stStationEvents[0].aEvents[18].bFault						:= TRUE;
stStationEvents[0].aEvents[18].bEventFlag					:= NOT stMachineStatus.bSystemPowerUp AND dw_T09_EL2809.stTerminalInfo.nTerminal_State <> 8;
stStationEvents[0].aEvents[18].bEventText					:= 'T09_EL2809 card in fault' ;
stStationEvents[0].aEvents[18].sSolution					:= 'Reset System';

(*stStationEvents[0].aEvents[19].bFault						:= TRUE;
stStationEvents[0].aEvents[19].bEventFlag					:= NOT stMachineStatus.bSystemPowerUp AND dw_T10_EL2809.stTerminalInfo.nTerminal_State <> 8;
stStationEvents[0].aEvents[19].bEventText					:= 'T10_EL2809 card in fault' ;
stStationEvents[0].aEvents[19].sSolution					:= 'Reset System';*)

stStationEvents[0].aEvents[20].bFault						:= TRUE;
stStationEvents[0].aEvents[20].bEventFlag					:= NOT stMachineStatus.bSystemPowerUp AND dw_T11_EL3058.stTerminalInfo.nTerminal_State <> 8;
stStationEvents[0].aEvents[20].bEventText					:= 'T11_EL3058 card in fault' ;
stStationEvents[0].aEvents[20].sSolution					:= 'Reset System';

stStationEvents[0].aEvents[22].bFault						:= TRUE;
stStationEvents[0].aEvents[22].bEventFlag					:= NOT stMachineStatus.bSystemPowerUp AND dw_T12_EL1918.stTerminalInfo.nTerminal_State <> 8;
stStationEvents[0].aEvents[22].bEventText					:= 'T12_EL1918 card in fault' ;
stStationEvents[0].aEvents[22].sSolution					:= 'Reset System';

stStationEvents[0].aEvents[23].bFault						:= TRUE;
stStationEvents[0].aEvents[23].bEventFlag					:= NOT stMachineStatus.bSystemPowerUp AND dw_T13_EL6633.stTerminalInfo.nTerminal_State <> 8;
stStationEvents[0].aEvents[23].bEventText					:= 'T13_EL6633 card in fault' ;
stStationEvents[0].aEvents[23].sSolution					:= 'Reset System';

stStationEvents[0].aEvents[24].bFault						:= TRUE;
stStationEvents[0].aEvents[24].bEventFlag					:= bDoorClosingFlag AND (NOT dw_T05_EL1918.iLeftTouchButtonNO OR NOT dw_T05_EL1918.iRightTouchButtonNO);
stStationEvents[0].aEvents[24].bEventText					:= 'Hands out before door was closed' ;
stStationEvents[0].aEvents[24].sSolution					:= 'Reset System';

stStationEvents[0].aEvents[25].bFault						:= TRUE;
stStationEvents[0].aEvents[25].bEventFlag					:= ((stMachineStatus.eMachineState = E_MachineState.MANUAL_MODE) OR (stMachineStatus.eMachineState = E_MachineState.SYSTEM_AUTO_CYCLE ))
																AND  NOT bHMIInitialized;
stStationEvents[0].aEvents[25].bEventText					:= 'Out HMI while Machine was in Autocycle' ;
stStationEvents[0].aEvents[25].sSolution					:= 'Reset System';


stStationEvents[0].aEvents[26].bFault						:= TRUE;
stStationEvents[0].aEvents[26].bEventTimer(IN := (stMachineStatus.eMachineState = E_MachineState.SYSTEM_AUTO_CYCLE) AND NOT bAutocycleIDLE, PT := stTimers.tAutoCycleTimeOut );
stStationEvents[0].aEvents[26].bEventFlag					:= stStationEvents[0].aEvents[26].bEventTimer.Q;
stStationEvents[0].aEvents[26].bEventText					:= 'Auto Cycle Timeout' ;
stStationEvents[0].aEvents[26].sSolution					:= 'Reset System';

//STOP REQUEST

stStationEvents[0].aEvents[40].bCycleStopRequest			:= TRUE;
stStationEvents[0].aEvents[40].bEventFlag					:= NOT bHMIInitialized;
stStationEvents[0].aEvents[40].bEventText					:= 'HMI not initialized' ;
stStationEvents[0].aEvents[40].sSolution					:= '';

stStationEvents[0].aEvents[41].bCycleStopRequest			:= TRUE;
stStationEvents[0].aEvents[41].bEventTimer(IN := bAutocycleIDLE, PT := stTimers.tAutoCycleIDLETimeOut);
stStationEvents[0].aEvents[41].bEventFlag					:= stStationEvents[0].aEvents[41].bEventTimer.Q;
stStationEvents[0].aEvents[41].bEventText					:= 'Autocycle in IDLE Timeout' ;
stStationEvents[0].aEvents[41].sSolution					:= '';

stStationEvents[0].aEvents[42].bCycleStopRequest			:= TRUE;
stStationEvents[0].aEvents[42].bEventFlag					:= NOT dw_T08_EL1809.iStopButton;
stStationEvents[0].aEvents[42].bEventText					:= 'Stop Button Pressed' ;
stStationEvents[0].aEvents[42].sSolution					:= '';
END_ACTION

END_PROGRAM

// ---- POUs/MAIN.TcPOU
PROGRAM MAIN
VAR
	
 
END_VAR

A_1_PRG_Main_Master();

END_PROGRAM

// ---- POUs/C_HMI/C_1_PRG_MainHMI.TcPOU
PROGRAM C_1_PRG_MainHMI
VAR
	
	bResetTest				: BOOL;
	i						: DINT;
	n						: DINT;//TABLE INDEX

END_VAR

a_ACT_MachineStatusBaner();
b_ACT_Timers();
c_ACT_IO();

bEnableSettings				:= (stMachineStatus.eMachineState = E_MachineState.STOPPED);

stStatisticsWH[0]			:= stStatisticsHMI[0];
stStatisticsWH[1]			:= stStatisticsHMI[3];
stStatisticsWH[2]			:= stStatisticsHMI[4];

stStatisticsLT[0]			:= stStatisticsHMI[0];
stStatisticsLT[1]			:= stStatisticsHMI[1];
stStatisticsLT[2]			:= stStatisticsHMI[2];

ACTION a_ACT_MachineStatusBaner:
//Machine status banner action
//SYSTEM POWER UP
IF stMachineStatus.bSystemPowerUp THEN	
	stStatusBanner.sMachineStatusText 							:= 'SYSTEM POWER UP';	
	stStatusBanner.nMachineStatusColour 						:= nWHITE;
	stStatusBanner.nMachineStatusTxtCol 						:= nBLACK;
	stStatusBanner.sBannerBckColor 								:= sWHITE;
	stStatusBanner.sBannerTextColor 							:= sBLACK;
END_IF

(* SYSTEM INITIALISING *)
IF stMachineStatus.bInitialising THEN	
	stStatusBanner.sMachineStatusText 							:= 'SYSTEM INITIALIZING';		
	stStatusBanner.nMachineStatusColour 						:= nYELLOW;
	stStatusBanner.nMachineStatusTxtCol 						:= nBLACK;
	stStatusBanner.sBannerBckColor 								:= sYELLOW;
	stStatusBanner.sBannerTextColor 							:= sBLACK;
END_IF

(* SAFETY *)
IF stMachineStatus.bSafety THEN	
	stStatusBanner.sMachineStatusText 							:= 'SYSTEM INITIALIZING';		
	stStatusBanner.nMachineStatusColour 						:= nYELLOW;
	stStatusBanner.nMachineStatusTxtCol 						:= nBLACK;
	stStatusBanner.sBannerBckColor 								:= sYELLOW;
	stStatusBanner.sBannerTextColor 							:= sBLACK;
END_IF


(* SYSTEM READY TO START FLASH ON *)
IF stMachineStatus.bReadyToStart AND stPuls.bFlash1Hz THEN
	stStatusBanner.sMachineStatusText 							:= 'SYSTEM READY TO START';		
	stStatusBanner.nMachineStatusColour 						:= nGREEN;
	stStatusBanner.nMachineStatusTxtCol 						:= nWHITE;
	stStatusBanner.sBannerBckColor 								:= sGREEN;
	stStatusBanner.sBannerTextColor 							:= sWHITE;
ELSIF stMachineStatus.bReadyToStart AND NOT stPuls.bFlash1Hz THEN	
	stStatusBanner.sMachineStatusText 							:= 'SYSTEM READY TO START';		
	stStatusBanner.nMachineStatusColour 						:= nWHITE;
	stStatusBanner.nMachineStatusTxtCol 						:= nGREEN;
	stStatusBanner.sBannerBckColor 								:= sWHITE;
	stStatusBanner.sBannerTextColor 							:= sGREEN;
END_IF

(* SYSTEM AUTO CYCLE *)
IF stMachineStatus.bAutoCycle THEN	
	stStatusBanner.sMachineStatusText 							:= 'SYSTEM AUTO CYCLE';		
	stStatusBanner.nMachineStatusColour 						:= nGREEN;
	stStatusBanner.nMachineStatusTxtCol 						:= nWHITE;
	stStatusBanner.sBannerBckColor 								:= sGREEN;
	stStatusBanner.sBannerTextColor 							:= sWHITE;	
END_IF

(* STOPPING *)
IF stMachineStatus.bStopping AND stPuls.bFlash1Hz THEN	
	stStatusBanner.sMachineStatusText 							:= 'STOPPING';		
	stStatusBanner.nMachineStatusColour 						:= nBLACK;
	stStatusBanner.nMachineStatusTxtCol 						:= nWHITE;
	stStatusBanner.sBannerBckColor 								:= sBLACK;
	stStatusBanner.sBannerTextColor 							:= sWHITE;	
ELSIF stMachineStatus.bStopping AND NOT stPuls.bFlash1Hz THEN	
	stStatusBanner.sMachineStatusText 							:= 'STOPPING';		
	stStatusBanner.nMachineStatusColour 						:= nWHITE;
	stStatusBanner.nMachineStatusTxtCol 						:= nBLACK;
	stStatusBanner.sBannerBckColor 								:= sWHITE;
	stStatusBanner.sBannerTextColor 							:= sBLACK;	
END_IF

(*STOPPED *)
IF stMachineStatus.bStopped THEN	
	stStatusBanner.sMachineStatusText 							:= 'CYCLE STOPPED';		
	stStatusBanner.nMachineStatusColour 						:= nBLACK;
	stStatusBanner.nMachineStatusTxtCol 						:= nWHITE;
	stStatusBanner.sBannerBckColor 								:= sBLACK;
	stStatusBanner.sBannerTextColor 							:= sWHITE;	
END_IF

(* FAULT FLASH ON *)
IF stMachineStatus.bFault AND stPuls.bFlash1Hz THEN	
	stStatusBanner.sMachineStatusText 							:= 'IMMEDIATE FAULT';		
	stStatusBanner.nMachineStatusColour 						:= nRED;
	stStatusBanner.nMachineStatusTxtCol 						:= nWHITE;
	stStatusBanner.sBannerBckColor 								:= sRED;
	stStatusBanner.sBannerTextColor 							:= sWHITE;	
ELSIF stMachineStatus.bFault AND NOT stPuls.bFlash1Hz THEN	
	stStatusBanner.sMachineStatusText 							:= 'IMMEDIATE FAULT';		
	stStatusBanner.nMachineStatusColour 						:= nWHITE;
	stStatusBanner.nMachineStatusTxtCol 						:= nBLACK;
	stStatusBanner.sBannerBckColor 								:= sWHITE;
	stStatusBanner.sBannerTextColor 							:= sBLACK;	
END_IF

(* MANUAL MODE *)
IF stMachineStatus.bManualMode THEN	
	stStatusBanner.sMachineStatusText 							:= 'MANUAL MODE';		
	stStatusBanner.nMachineStatusColour 						:= nBLUE;
	stStatusBanner.nMachineStatusTxtCol 						:= nWHITE;
	stStatusBanner.sBannerBckColor 								:= sBLUE;
	stStatusBanner.sBannerTextColor 							:= sWHITE;	
END_IF
END_ACTION

ACTION b_ACT_Timers:

stTimers.tAutoCycleTimeOut		:= DINT_TO_TIME(stTimers.nAutoCycleTimeOut * 1000) ;
stTimers.tDoorOpenedSignal		:= DINT_TO_TIME(stTimers.nDoorOpenedSignal * 1000) ;
stTimers.tStation1TimeOut		:= DINT_TO_TIME(stTimers.nStation1TimeOut * 1000) ;
stTimers.tStation2TimeOut		:= DINT_TO_TIME(stTimers.nStation2TimeOut * 1000) ;
stTimers.tStation3TimeOut		:= DINT_TO_TIME(stTimers.nStation3TimeOut * 1000) ;
stTimers.tTwoHandsSignal		:= DINT_TO_TIME(stTimers.nTwoHandsSignal * 1000) ;
stTimers.tHeightTest			:= DINT_TO_TIME(stTimers.nHeightTest * 1000) ;
stTimers.tAutoCycleIDLETimeOut			:= DINT_TO_TIME(stTimers.nAutoCycleIDLETimeOut * 1000) ;
END_ACTION

ACTION c_ACT_IO:


bLeftHand							:= dw_T05_EL1918.iLeftTouchButtonNO;
bRightHand							:= dw_T05_EL1918.iRightTouchButtonNO;
END_ACTION

END_PROGRAM

// ---- POUs/B_STATIONS/B_2_HEIGHT_TEST/B_2_1_PRG_Master_Height_Test.TcPOU
PROGRAM B_2_1_PRG_Master_Height_Test

VAR

	rGoodStatistics						: ARRAY[0..1] OF  R_TRIG;
	rBadStatistics						: ARRAY[0..1] OF  R_TRIG;
	rEfficency							: STRING(510);
	
	anMinimumDistance					: ARRAY[1..3] OF REAL;
	anMaximumDistance					: ARRAY[1..3] OF REAL;

/////////////////////////////////////////////////////////////////////////////////////I O/////////////////////////////////////////////////////////////////////////////////////	
	
	abPass1								: ARRAY [1..3] OF BOOL;
	abFail1								: ARRAY [1..3] OF BOOL;
	abPass2								: ARRAY [1..3] OF BOOL;
	abFail2								: ARRAY [1..3] OF BOOL;
	tonTakeMeasure						: TON;
	abMeaurement						: ARRAY [0..1] OF BOOL;
	bMeasurementDone					: BOOL;

	abProbeError1						: ARRAY[1..4] OF BOOL;
	abProbeError2						: ARRAY[1..4] OF BOOL;
	bGeneralProbeError					: BOOL;
	bGeneralError						: BOOL;
	anRawMesurement1					: ARRAY[1..4] OF REAL;
	anRawMesurement2					: ARRAY[1..4] OF REAL;
	anRealDistance1						: ARRAY[1..3] OF REAL;
	anRealDistance2						: ARRAY[1..3] OF REAL;
	

	
	i									: DINT;
	j									: DINT; //Index for settings
	
	
	

	
END_VAR

d_ACT_Set_Events_Station_2();
a_ACT_Ctrl_Station_2();
b_ACT_IO();
c_ACT_Statistics_Station_2();
e_ACT_Measurement();
f_ACT_ManualMode();
g_ACT_Settings();

ACTION a_ACT_Ctrl_Station_2:
/////////////////////////////////////////////////////////////////////////////////////UTILITIES/////////////////////////////////////////////////////////////////////////////////////
IF bGeneralProbeError OR bGeneralError OR stHeightTests.CMD.bAbort THEN
	
	stHeightTests.State			:= E_HeightTest_State.RESET;

ELSIF stHeightTests.CMD.bManualMode THEN
	
	stHeightTests.State			:= E_HeightTest_State.MANUAL_MODE;
	
END_IF



/////////////////////////////////////////////////////////////////////////////////////CONDITIONS/////////////////////////////////////////////////////////////////////////////////////

CASE stHeightTests.State OF
	
	E_HeightTest_State.ABORTED:

								IF 	stHeightTests.CMD.bEnable THEN
									
									stHeightTests.State			:= E_HeightTest_State.READY;
								
								END_IF
								
								

	E_HeightTest_State.READY:
	
								IF stHeightTests.CMD.bExecute THEN
									
									stHeightTests.State			:= E_HeightTest_State.MEASURE;
								
								END_IF
		
	E_HeightTest_State.MEASURE:				
									
								IF stHeightTests.CMD.HeightTest_CMD.Measurement1 AND stHeightTests.CMD.HeightTest_CMD.Measurement2 THEN
										
									abMeaurement[0]			:= TRUE;
									abMeaurement[1]			:= TRUE;
									
								ELSIF stHeightTests.CMD.HeightTest_CMD.Measurement1 AND NOT stHeightTests.CMD.HeightTest_CMD.Measurement2 THEN
									
									abMeaurement[0]			:= TRUE;
									
								ELSIF NOT stHeightTests.CMD.HeightTest_CMD.Measurement1 AND stHeightTests.CMD.HeightTest_CMD.Measurement2 THEN
									
									abMeaurement[1]			:= TRUE;
									
								END_IF
									
								stHeightTests.State			:= E_HeightTest_State.WAIT_MEASUREMENT;
								
	E_HeightTest_State.WAIT_MEASUREMENT:						
								
								e_ACT_Measurement();
								
								IF stHeightTests.CMD.HeightTest_CMD.Measurement1 THEN
									
									stCycleDataNest1.HeightTest_anRawMeasurement				:= anRawMesurement1;
									stCycleDataNest1.HeightTest_anDistancesResult 				:= anRealDistance1;
									stCycleDataNest1.HeightTest_bDistancesResult				:= abPass1;
									
								END_IF
								IF stHeightTests.CMD.HeightTest_CMD.Measurement2 THEN
									
									stCycleDataNest2.HeightTest_anRawMeasurement				:= anRawMesurement2;																
									stCycleDataNest2.HeightTest_anDistancesResult 				:= anRealDistance2;																
									stCycleDataNest2.HeightTest_bDistancesResult				:= abPass2;
									
								END_IF
								
								
								IF bMeasurementDone THEN
			
									stHeightTests.State		:= E_HeightTest_State.DONE;
								
								END_IF
										
	E_HeightTest_State.DONE:
								IF  stHeightTests.CMD.bAcknowledge THEN
									
									stHeightTests.State									:= E_HeightTest_State.RESULTS;
									stHeightTests.CMD.bAcknowledge 						:= FALSE;
									
								END_IF	
								
	E_HeightTest_State.RESULTS:
							
								IF abMeaurement[0] THEN
									IF abPass1[1] AND abPass1[2] AND abPass1[3] THEN
									
										stCycleDataNest1.HeightTest_Pass				:= TRUE;
									
									ELSE stCycleDataNest1.HeightTest_Fail 				:= TRUE;
								
									END_IF
								END_IF
								
								IF abMeaurement[1] THEN
									IF abPass2[1] AND abPass2[2] AND abPass2[3] THEN
									
										stCycleDataNest2.HeightTest_Pass				:= TRUE;
									
									ELSE stCycleDataNest2.HeightTest_Fail  			:= TRUE;
								
									END_IF
								END_IF	
								
								stHeightTests.State										:= E_HeightTest_State.RESET;
								
	E_HeightTest_State.RESET:
	
								abMeaurement[0]											:= FALSE;
								abMeaurement[1]											:= FALSE;
								bMeasurementDone										:= FALSE;

								FOR i := 1 TO 3 DO
									
									abPass1[i]											:= FALSE;
									abFail1[i]											:= FALSE;
									abPass2[i]											:= FALSE;
									abFail2[i]											:= FALSE;
								
								END_FOR
								
								IF bGeneralProbeError OR bGeneralError THEN
									
									stHeightTests.State									:= E_HeightTest_State.ERROR;
								
								ELSIF stHeightTests.CMD.bAbort THEN
									
									stHeightTests.State									:= E_HeightTest_State.ABORTED;
								
								ELSE stHeightTests.State								:= E_HeightTest_State.READY;
									
								END_IF
								
								
	
	E_HeightTest_State.ERROR:
	
								IF NOT bGeneralProbeError OR bGeneralError THEN
									
									stHeightTests.State									:= E_HeightTest_State.RESET;
									
								END_IF
							
	E_HeightTest_State.MANUAL_MODE:
	
								f_ACT_ManualMode();
								
								IF NOT stHeightTests.CMD.bManualMode THEN
									
									stHeightTests.State									:= E_HeightTest_State.ABORTED;
									
								END_IF
								
	
								

ELSE stHeightTests.State := E_HeightTest_State.READY;
	
END_CASE
/////////////////////////////////////////////////////////////////////////////////////STATUS/////////////////////////////////////////////////////////////////////////////////////

stHeightTests.Status.bBusy	:= 	stHeightTests.State	= E_HeightTest_State.WAIT_MEASUREMENT;	

stHeightTests.Status.bDone	:= 	stHeightTests.State	= E_HeightTest_State.DONE;

stHeightTests.Status.bError	:= 	stHeightTests.State	= E_HeightTest_State.ERROR;	

stHeightTests.Status.bReady	:=	stHeightTests.State	= E_HeightTest_State.READY;

stHeightTests.Status.bStopped := NOT stHeightTests.Status.bBusy;
END_ACTION

ACTION b_ACT_IO:

	abProbeError1					:= Probes.stProbesSet[1].abProbeError;
	abProbeError2					:= Probes.stProbesSet[2].abProbeError;
	bGeneralError					:= Probes.bGeneralError;
	anRawMesurement1				:= Probes.stProbesSet[1].anScaledRawMeasurement;
	anRawMesurement2				:= Probes.stProbesSet[2].anScaledRawMeasurement;
	


	bGeneralProbeError				:= 	abProbeError1[1] OR abProbeError1[2] OR abProbeError1[3] OR abProbeError1[4] OR
										abProbeError2[1] OR abProbeError2[2] OR abProbeError2[3] OR abProbeError2[4];
										
	stCycleDataNest1.HeightTest_anSetPoint := stProbesSettings.anExpectedDistances;
	stCycleDataNest2.HeightTest_anSetPoint := stProbesSettings.anExpectedDistances;
END_ACTION

ACTION c_ACT_Statistics_Station_2:
stStatisticsHMI[3].sName			:= 'Height Test 1';
stStatisticsHMI[4].sName			:= 'Height Test 2';


rGoodStatistics[0]( CLK := stCycleDataNest1.HeightTest_Pass);
rGoodStatistics[1]( CLK := stCycleDataNest2.HeightTest_Pass);
rBadStatistics[0]	( CLK := stCycleDataNest1.HeightTest_Fail);
rBadStatistics[1]	( CLK := stCycleDataNest2.HeightTest_Fail);

//statistics 1
IF 	rGoodStatistics[0].Q THEN
	
	stStatisticsHMI[3].nGood		:= stStatisticsHMI[3].nGood + 1;
	stStatisticsHMI[3].nTotalGood	:= stStatisticsHMI[3].nTotalGood + 1;
	
END_IF
								
IF 	rBadStatistics[0].Q THEN
	
	stStatisticsHMI[3].nBad			:= stStatisticsHMI[3].nBad + 1;
	stStatisticsHMI[3].nTotalBad	:= stStatisticsHMI[3].nTotalBad + 1;
	
END_IF

IF stStatisticsHMI[3].bResetGood THEN
	stStatisticsHMI[3].nGood		:= 0;
END_IF

IF stStatisticsHMI[3].bResetBad THEN
	stStatisticsHMI[3].nBad			:= 0;
END_IF

IF (( stStatisticsHMI[3].nGood + stStatisticsHMI[3].nBad) <> 0) THEN
	
	rEfficency							:= LREAL_TO_FMTSTR(in := (DINT_TO_REAL(stStatisticsHMI[3].nGood) /( DINT_TO_REAL(stStatisticsHMI[3].nGood) + DINT_TO_REAL(stStatisticsHMI[3].nBad))) * 100.0,iPrecision := 2, bRound := TRUE);
	stStatisticsHMI[3].nEfficency		:= CONCAT(STR1 := '%', STR2 := (rEfficency));

ELSE stStatisticsHMI[3].nEfficency		:= CONCAT(STR1 := '%', STR2 := (DINT_TO_STRING(0)));
	
END_IF
//statistics 2
IF 	rGoodStatistics[1].Q THEN
	
	stStatisticsHMI[4].nGood		:= stStatisticsHMI[4].nGood + 1;
	stStatisticsHMI[4].nTotalGood	:= stStatisticsHMI[4].nTotalGood + 1;
	
END_IF
								
IF 	rBadStatistics[1].Q THEN
	
	stStatisticsHMI[4].nBad			:= stStatisticsHMI[4].nBad + 1;
	stStatisticsHMI[4].nTotalBad	:= stStatisticsHMI[4].nTotalBad + 1;
	
END_IF

IF stStatisticsHMI[4].bResetGood THEN
	stStatisticsHMI[4].nGood		:= 0;
END_IF

IF stStatisticsHMI[4].bResetBad THEN
	stStatisticsHMI[4].nBad			:= 0;
END_IF

IF (( stStatisticsHMI[4].nGood + stStatisticsHMI[4].nBad) <> 0) THEN
	
	rEfficency							:= LREAL_TO_FMTSTR(in := (DINT_TO_REAL(stStatisticsHMI[4].nGood) /( DINT_TO_REAL(stStatisticsHMI[4].nGood) + DINT_TO_REAL(stStatisticsHMI[4].nBad))) * 100.0,iPrecision := 2, bRound := TRUE);
	stStatisticsHMI[4].nEfficency		:= CONCAT(STR1 := '%', STR2 := (rEfficency));

ELSE stStatisticsHMI[4].nEfficency		:= CONCAT(STR1 := '%', STR2 := (DINT_TO_STRING(0)));
	
END_IF
END_ACTION

ACTION d_ACT_Set_Events_Station_2:
//FAULTS

stStationEvents[2].aEvents[0].bFault						:= TRUE;
stStationEvents[2].aEvents[0].bEventFlag					:= bGeneralError;
stStationEvents[2].aEvents[0].bEventText					:= 'Probes general error';
stStationEvents[2].aEvents[0].sSolution						:= 'Check probes amplifier and ethercat unit';

stStationEvents[2].aEvents[1].bFault						:= TRUE;
stStationEvents[2].aEvents[1].bEventFlag					:= abProbeError1[1];
stStationEvents[2].aEvents[1].bEventText					:= 'Probes 1 error';
stStationEvents[2].aEvents[1].sSolution						:= 'Check probe 1';

stStationEvents[2].aEvents[2].bFault						:= TRUE;
stStationEvents[2].aEvents[2].bEventFlag					:= abProbeError1[2];
stStationEvents[2].aEvents[2].bEventText					:= 'Probes 2 error';
stStationEvents[2].aEvents[2].sSolution						:= 'Check probe 2';

stStationEvents[2].aEvents[3].bFault						:= TRUE;
stStationEvents[2].aEvents[3].bEventFlag					:= abProbeError1[3];
stStationEvents[2].aEvents[3].bEventText					:= 'Probes 3 error';
stStationEvents[2].aEvents[3].sSolution						:= 'Check probe 3';

stStationEvents[2].aEvents[4].bFault						:= TRUE;
stStationEvents[2].aEvents[4].bEventFlag					:= abProbeError1[4];
stStationEvents[2].aEvents[4].bEventText					:= 'Probes 4 error';
stStationEvents[2].aEvents[4].sSolution						:= 'Check probe 4';

stStationEvents[2].aEvents[5].bFault						:= TRUE;
stStationEvents[2].aEvents[5].bEventFlag					:= abProbeError2[1];
stStationEvents[2].aEvents[5].bEventText					:= 'Probes 5 error';
stStationEvents[2].aEvents[5].sSolution						:= 'Check probe 5';

stStationEvents[2].aEvents[6].bFault						:= TRUE;
stStationEvents[2].aEvents[6].bEventFlag					:= abProbeError2[2];
stStationEvents[2].aEvents[6].bEventText					:= 'Probes 6 error';
stStationEvents[2].aEvents[6].sSolution						:= 'Check probe 6';

stStationEvents[2].aEvents[7].bFault						:= TRUE;
stStationEvents[2].aEvents[7].bEventFlag					:= abProbeError2[3];
stStationEvents[2].aEvents[7].bEventText					:= 'Probes 7 error';
stStationEvents[2].aEvents[7].sSolution						:= 'Check probe 7';

stStationEvents[2].aEvents[8].bFault						:= TRUE;
stStationEvents[2].aEvents[8].bEventFlag					:= abProbeError2[4];
stStationEvents[2].aEvents[8].bEventText					:= 'Probes 8 error';
stStationEvents[2].aEvents[8].sSolution						:= 'Check probe 8';

stStationEvents[2].aEvents[9].bFault						:= TRUE;
stStationEvents[2].aEvents[9].bEventTimer(IN := stHeightTests.Status.bBusy, PT := stTimers.tStation2TimeOut);
stStationEvents[2].aEvents[9].bEventFlag					:= stStationEvents[2].aEvents[9].bEventTimer.Q;
stStationEvents[2].aEvents[9].bEventText					:= 'Height test cycle Timeout';
stStationEvents[2].aEvents[9].sSolution						:= 'Reset System';

(*//CYCLE STOP FAULT

stStationEvents[2].aEvents[1].bFault						:= TRUE;
stStationEvents[2].aEvents[1].bEventFlag					:= bEventsFlag[1];
stStationEvents[2].aEvents[1].bEventText					:= 'ST1 EVENT 1';
stStationEvents[2].aEvents[1].sSolution						:= 'Solution 4';


//CYCLE STOP REQUEST

stStationEvents[2].aEvents[2].bCycleStopRequest				:= TRUE;
stStationEvents[2].aEvents[2].bEventFlag					:= bEventsFlag[2];
stStationEvents[2].aEvents[2].bEventText					:= 'ST1 EVENT 2';*)
END_ACTION

ACTION e_ACT_Measurement:

tonTakeMeasure(IN:= stHeightTests.State = E_HeightTest_State.WAIT_MEASUREMENT, PT := stTimers.tHeightTest);

IF tonTakeMeasure.Q THEN
	
	IF abMeaurement[0] THEN
	
		FOR i := 1 TO 3 DO
		
			IF (anRealDistance1[i] > anMinimumDistance[i]) AND (anRealDistance1[i] < anMaximumDistance[i]) THEN
		
				abPass1[i]						:= TRUE;
			
			ELSE abFail1[i]						:= TRUE;	
				
			END_IF
		
		END_FOR

	END_IF
	
	IF abMeaurement[1] THEN
	
		FOR i := 1 TO 3 DO
		
			IF (anRealDistance2[i] > anMinimumDistance[i]) AND (anRealDistance2[i] < anMaximumDistance[i]) THEN
		
				abPass2[i]						:= TRUE;
			
			ELSE abFail2[i]						:= TRUE;	
				
			END_IF
		
		END_FOR

	END_IF

	bMeasurementDone							:= TRUE;
	i											:= 0;
END_IF
END_ACTION

ACTION f_ACT_ManualMode:
IF stPuls.bFlash100Hz THEN
	
	FOR i := 1 TO 3 DO
		
		IF (anRealDistance1[i] > anMinimumDistance[i]) AND (anRealDistance1[i] < anMaximumDistance[i]) THEN
		
			stAnimations.abDistanceBoxesGreen[i]	:= TRUE;
			
		ELSE stAnimations.abDistanceBoxesGreen[i]	:= FALSE;	
				
		END_IF
		
	END_FOR
	i												:= 0;
	FOR i := 1 TO 3 DO
		
		IF (anRealDistance2[i] > anMinimumDistance[i]) AND (anRealDistance2[i] < anMaximumDistance[i]) THEN
		
			stAnimations.abDistanceBoxesGreen[3+i]	:= TRUE;
			
		ELSE stAnimations.abDistanceBoxesGreen[3+i]	:= FALSE;	
				
		END_IF
		
	END_FOR
	
	i												:= 0;
END_IF
END_ACTION

ACTION g_ACT_Settings:
//settings tolerances

anMinimumDistance[1]					:= stProbesSettings.anExpectedDistances[1] - stProbesSettings.anTolerances[1];//settings from HMI
anMaximumDistance[1]					:= stProbesSettings.anExpectedDistances[1] + stProbesSettings.anTolerances[1];//settings from HMI
anMinimumDistance[2]					:= stProbesSettings.anExpectedDistances[2] - stProbesSettings.anTolerances[2];//settings from HMI
anMaximumDistance[2]					:= stProbesSettings.anExpectedDistances[2] + stProbesSettings.anTolerances[2];//settings from HMI
anMinimumDistance[3]					:= stProbesSettings.anExpectedDistances[3] - stProbesSettings.anTolerances[3];//settings from HMI
anMaximumDistance[3]					:= stProbesSettings.anExpectedDistances[3] + stProbesSettings.anTolerances[3];//settings from HMI





//setting the bit according to the probe from bit 1 to bit 8
IF abPresetProbe[1] THEN
	
	Probes.abPresetProbe						:= 2;

ELSIF abPresetProbe[2] THEN
	
	Probes.abPresetProbe						:= 4;
	
ELSIF abPresetProbe[3] THEN
	
	Probes.abPresetProbe						:= 8;
	
ELSIF abPresetProbe[4] THEN
	
	Probes.abPresetProbe						:= 16;
	
ELSIF abPresetProbe[5] THEN
	
	Probes.abPresetProbe						:= 32;
	
ELSIF abPresetProbe[6] THEN
	
	Probes.abPresetProbe						:= 64;
	
ELSIF abPresetProbe[7] THEN
	
	Probes.abPresetProbe						:= 128;
	
ELSIF abPresetProbe[8] THEN
	
	Probes.abPresetProbe						:= 256;

END_IF

Probes.stProbesSet[1].anScaledRawMeasurement[1]					:= DINT_TO_REAL(Probes.stProbesSet[1].anRawMeasurement[1])/10000;
Probes.stProbesSet[1].anScaledRawMeasurement[2]					:= DINT_TO_REAL(Probes.stProbesSet[1].anRawMeasurement[2])/10000;
Probes.stProbesSet[1].anScaledRawMeasurement[3]					:= DINT_TO_REAL(Probes.stProbesSet[1].anRawMeasurement[3])/10000;
Probes.stProbesSet[1].anScaledRawMeasurement[4]					:= DINT_TO_REAL(Probes.stProbesSet[1].anRawMeasurement[4])/10000;

Probes.stProbesSet[2].anScaledRawMeasurement[1]					:= DINT_TO_REAL(Probes.stProbesSet[2].anRawMeasurement[1])/10000;
Probes.stProbesSet[2].anScaledRawMeasurement[2]					:= DINT_TO_REAL(Probes.stProbesSet[2].anRawMeasurement[2])/10000;
Probes.stProbesSet[2].anScaledRawMeasurement[3]					:= DINT_TO_REAL(Probes.stProbesSet[2].anRawMeasurement[3])/10000;
Probes.stProbesSet[2].anScaledRawMeasurement[4]					:= DINT_TO_REAL(Probes.stProbesSet[2].anRawMeasurement[4])/10000;

IF Probes.stProbesSet[1].anScaledRawMeasurement[1] > 4 AND Probes.stProbesSet[1].anScaledRawMeasurement[1] < 8 AND 
	Probes.stProbesSet[1].anScaledRawMeasurement[2] > 4 AND Probes.stProbesSet[1].anScaledRawMeasurement[2] < 8 AND 
	Probes.stProbesSet[1].anScaledRawMeasurement[3] > 4 AND Probes.stProbesSet[1].anScaledRawMeasurement[3] < 8 AND 
	Probes.stProbesSet[1].anScaledRawMeasurement[4] > 4 AND Probes.stProbesSet[1].anScaledRawMeasurement[4] < 8 THEN 
	
	bEnableSetCablibrationBlock1								:= TRUE;
	
ELSE bEnableSetCablibrationBlock1								:= FALSE;
	
END_IF

IF Probes.stProbesSet[2].anScaledRawMeasurement[1] > 4 AND Probes.stProbesSet[2].anScaledRawMeasurement[1] < 8 AND 
	Probes.stProbesSet[2].anScaledRawMeasurement[2] > 4 AND Probes.stProbesSet[2].anScaledRawMeasurement[2] < 8 AND 
	Probes.stProbesSet[2].anScaledRawMeasurement[3] > 4 AND Probes.stProbesSet[2].anScaledRawMeasurement[3] < 8 AND 
	Probes.stProbesSet[2].anScaledRawMeasurement[4] > 4 AND Probes.stProbesSet[2].anScaledRawMeasurement[4] < 8 THEN 
	
	bEnableSetCablibrationBlock2								:= TRUE;
	
ELSE bEnableSetCablibrationBlock2								:= FALSE;
	
END_IF

//calibration block
IF bSetCalibrationBlock1 THEN
	
	stProbesSettings.anHeightSetByCalibration1[1]				:= Probes.stProbesSet[1].anScaledRawMeasurement[1];
	stProbesSettings.anHeightSetByCalibration1[2]				:= Probes.stProbesSet[1].anScaledRawMeasurement[2];
	stProbesSettings.anHeightSetByCalibration1[3]				:= Probes.stProbesSet[1].anScaledRawMeasurement[3];
	stProbesSettings.anHeightSetByCalibration1[4]				:= Probes.stProbesSet[1].anScaledRawMeasurement[4];
	
	stProbesSettings.nDistanceOffset1[1]						:= stProbesSettings.anDistanceCalibrationBlock[1] - (Probes.stProbesSet[1].anScaledRawMeasurement[2] - Probes.stProbesSet[1].anScaledRawMeasurement[1]);
	stProbesSettings.nDistanceOffset1[2]						:= stProbesSettings.anDistanceCalibrationBlock[2] - (Probes.stProbesSet[1].anScaledRawMeasurement[3] - Probes.stProbesSet[1].anScaledRawMeasurement[1]);
	stProbesSettings.nDistanceOffset1[3]						:= stProbesSettings.anDistanceCalibrationBlock[3] - (Probes.stProbesSet[1].anScaledRawMeasurement[4] - Probes.stProbesSet[1].anScaledRawMeasurement[1]);
	
END_IF

IF bSetCalibrationBlock2 THEN
	
	stProbesSettings.anHeightSetByCalibration2[1]				:= Probes.stProbesSet[2].anScaledRawMeasurement[1];
	stProbesSettings.anHeightSetByCalibration2[2]				:= Probes.stProbesSet[2].anScaledRawMeasurement[2];
	stProbesSettings.anHeightSetByCalibration2[3]				:= Probes.stProbesSet[2].anScaledRawMeasurement[3];
	stProbesSettings.anHeightSetByCalibration2[4]				:= Probes.stProbesSet[2].anScaledRawMeasurement[4];
	
	stProbesSettings.nDistanceOffset2[1]						:= stProbesSettings.anDistanceCalibrationBlock[1] - (Probes.stProbesSet[2].anScaledRawMeasurement[2] - Probes.stProbesSet[2].anScaledRawMeasurement[1]);
	stProbesSettings.nDistanceOffset2[2]						:= stProbesSettings.anDistanceCalibrationBlock[2] - (Probes.stProbesSet[2].anScaledRawMeasurement[3] - Probes.stProbesSet[2].anScaledRawMeasurement[1]);
	stProbesSettings.nDistanceOffset2[3]						:= stProbesSettings.anDistanceCalibrationBlock[3] - (Probes.stProbesSet[2].anScaledRawMeasurement[4] - Probes.stProbesSet[2].anScaledRawMeasurement[1]);

END_IF

anRealDistance1[1] 								:= (Probes.stProbesSet[1].anScaledRawMeasurement[2] - Probes.stProbesSet[1].anScaledRawMeasurement[1]) + stProbesSettings.nDistanceOffset1[1];
anRealDistance1[2] 								:= (Probes.stProbesSet[1].anScaledRawMeasurement[3] - Probes.stProbesSet[1].anScaledRawMeasurement[1]) + stProbesSettings.nDistanceOffset1[2];
anRealDistance1[3] 								:= (Probes.stProbesSet[1].anScaledRawMeasurement[4] - Probes.stProbesSet[1].anScaledRawMeasurement[1]) + stProbesSettings.nDistanceOffset1[3];

anRealDistance2[1] 								:= (Probes.stProbesSet[2].anScaledRawMeasurement[2] - Probes.stProbesSet[2].anScaledRawMeasurement[1]) + stProbesSettings.nDistanceOffset2[1];
anRealDistance2[2] 								:= (Probes.stProbesSet[2].anScaledRawMeasurement[3] - Probes.stProbesSet[2].anScaledRawMeasurement[1]) + stProbesSettings.nDistanceOffset2[2];
anRealDistance2[3] 								:= (Probes.stProbesSet[2].anScaledRawMeasurement[4] - Probes.stProbesSet[2].anScaledRawMeasurement[1]) + stProbesSettings.nDistanceOffset2[3];
END_ACTION

END_PROGRAM

// ---- POUs/B_STATIONS/B_1_LEAK_TEST/B_1_1_PRG_Master_Leak_Test.TcPOU
PROGRAM B_1_1_PRG_Master_Leak_Test

VAR

	tonStationStopped					: TON;
	tonExecute							: TON;
	rGoodStatistics						: ARRAY [0..1] OF R_TRIG;
	rBadStatistics						: ARRAY [0..1] OF R_TRIG;
	rEfficency							: ARRAY [0..1] OF STRING(510);
	
	tonWaitResults						: TON;
/////////////////////////////////////////////////////////////////////////////////////I O/////////////////////////////////////////////////////////////////////////////////////	

	bStopped							: ARRAY [0..1] OF BOOL;
	bError								: ARRAY [0..1] OF BOOL;
	bReady								: ARRAY [0..1] OF BOOL;
	bDone								: ARRAY [0..1] OF BOOL;
	bReset								: ARRAY [0..1] OF BOOL;
	bStart								: ARRAY [0..1] OF BOOL;
	bStop								: ARRAY [0..1] OF BOOL;	
	bBusy								: ARRAY [0..1] OF BOOL;	
	fLeakTestDone						: ARRAY [0..1] OF F_TRIG;	
	bLeakTestDone						: ARRAY [0..1] OF BOOL;	
	rPass								: ARRAY [0..1] OF R_TRIG;	
	bPass								: ARRAY [0..1] OF BOOL;	
	rFail								: ARRAY [0..1] OF R_TRIG;	
	bFail								: ARRAY [0..1] OF BOOL;
	rReset								: ARRAY [0..1] OF R_TRIG;

	
END_VAR

a_ACT_Ctrl_Station_1();
b_ACT_IO();
c_ACT_Statistics_Station_1();
d_ACT_Set_Events_Station_1();

ACTION a_ACT_Ctrl_Station_1:
/////////////////////////////////////////////////////////////////////////////////////UTILITIES/////////////////////////////////////////////////////////////////////////////////////
tonStationStopped( IN := bStopped[0] AND bStopped[1], PT := T#1S);
tonExecute(IN := stLeakTesters.State = E_LeakTester_State.RUN_LEAK_TESTERS, PT := T#500MS);
tonWaitResults(IN := (stLeakTesters.State = E_LeakTester_State.WAIT_RESULTS), PT := T#100MS);

/////////////////////////////////////////////////////////////////////////////////////CONDITIONS/////////////////////////////////////////////////////////////////////////////////////

IF stLeakTesters.CMD.bAbort OR bError[0] OR bError[1] THEN
								
	stLeakTesters.State											:= E_LeakTester_State.RESET;
	

END_IF



CASE stLeakTesters.State OF
	
	E_LeakTester_State.ABORTED:
	
								IF stLeakTesters.CMD.bEnable AND NOT bError[0] THEN
									stLeakTesters.State			:= E_LeakTester_State.HOMING;
								ELSIF bError[0] OR bError[1] THEN
									stLeakTesters.State			:= E_LeakTester_State.ERROR;
								END_IF
	
	E_LeakTester_State.HOMING:
	
								IF bReady[0] AND bReady[1] AND bStopped[0] AND bStopped[1] THEN
									stLeakTesters.State			:= E_LeakTester_State.READY;
								
								END_IF
								
	E_LeakTester_State.READY:
	
								IF stLeakTesters.CMD.bExecute THEN
									
									stLeakTesters.State			:= E_LeakTester_State.RUN_LEAK_TESTERS;
								
								END_IF
		
								
	E_LeakTester_State.RUN_LEAK_TESTERS:	
								
								IF stLeakTesters.CMD.LeakTestersCMD.RunLeakTester1 AND stLeakTesters.CMD.LeakTestersCMD.RunLeakTester2 THEN
										
										bStart[0]				:= TRUE;
										bStart[1]				:= TRUE;
									
								ELSIF stLeakTesters.CMD.LeakTestersCMD.RunLeakTester1 AND NOT stLeakTesters.CMD.LeakTestersCMD.RunLeakTester2 THEN
										
										bStart[0]				:= TRUE;
									
								ELSIF NOT stLeakTesters.CMD.LeakTestersCMD.RunLeakTester1 AND stLeakTesters.CMD.LeakTestersCMD.RunLeakTester2 THEN
										
										bStart[1]				:= TRUE;
									
								END_IF
								
								IF tonExecute.Q THEN
									
									stLeakTesters.State			:= E_LeakTester_State.WAIT_LEAK_TESTERS;
								
								END_IF
	
	E_LeakTester_State.WAIT_LEAK_TESTERS:
	
								IF stLeakTesters.CMD.LeakTestersCMD.RunLeakTester1 AND stLeakTesters.CMD.LeakTestersCMD.RunLeakTester2 THEN
										
										IF bLeakTestDone[0] AND bLeakTestDone[1] THEN
											
											stLeakTesters.State	:= E_LeakTester_State.WAIT_RESULTS;
											
										END_IF
									
								ELSIF stLeakTesters.CMD.LeakTestersCMD.RunLeakTester1 AND NOT stLeakTesters.CMD.LeakTestersCMD.RunLeakTester2 THEN
										
										IF bLeakTestDone[0]  THEN
											
											stLeakTesters.State	:= E_LeakTester_State.WAIT_RESULTS;
											
										END_IF
									
								ELSIF NOT stLeakTesters.CMD.LeakTestersCMD.RunLeakTester1 AND stLeakTesters.CMD.LeakTestersCMD.RunLeakTester2 THEN
										
										IF bLeakTestDone[1]  THEN
											
											stLeakTesters.State	:= E_LeakTester_State.WAIT_RESULTS;
											
										END_IF
									
								END_IF
	
	E_LeakTester_State.WAIT_RESULTS:
	
								IF tonWaitResults.Q THEN
									
									stLeakTesters.State	:= E_LeakTester_State.RESULTS;
									
								END_IF


		
	E_LeakTester_State.RESULTS:
								
								IF stLeakTesters.CMD.LeakTestersCMD.RunLeakTester1 THEN
									
									IF bPass[0] THEN
									
										stCycleDataNest1.LeakTest_Pass := TRUE;
										stCycleDataNest1.LeakTest_Fail := FALSE;
										
										stLeakTesters.State	:= E_LeakTester_State.DONE;
								
									ELSIF bFail[0] THEN
									
										stCycleDataNest1.LeakTest_Fail := TRUE;
										stCycleDataNest1.LeakTest_Pass := FALSE;
								
										stLeakTesters.State	:= E_LeakTester_State.DONE;
										
								END_IF
									
								END_IF
								
								IF stLeakTesters.CMD.LeakTestersCMD.RunLeakTester2 THEN
									
									IF bPass[1] THEN
									
										stCycleDataNest2.LeakTest_Pass := TRUE;
										stCycleDataNest2.LeakTest_Fail	:= FALSE;
										
										stLeakTesters.State	:= E_LeakTester_State.DONE;
								
									ELSIF bFail[1] THEN
									
										stCycleDataNest2.LeakTest_Fail	:= TRUE;
										stCycleDataNest2.LeakTest_Pass := FALSE;
										
										stLeakTesters.State	:= E_LeakTester_State.DONE;
								
								END_IF
									
								END_IF
								
								
								
		E_LeakTester_State.DONE:
								IF  stLeakTesters.CMD.bAcknowledge THEN
									
									stLeakTesters.CMD.bAcknowledge := FALSE;
									stLeakTesters.State			:= E_LeakTester_State.RESET;
									
								END_IF	
								
								
								
	E_LeakTester_State.RESET:
	

								bStart[0]						:= FALSE;
								bStart[1]						:= FALSE;
								bReset[0]						:= FALSE;
								bReset[1]						:= FALSE;
								bStop[0]						:= FALSE;
								bStop[1]						:= FALSE;
								bLeakTestDone[0]				:= FALSE;
								bLeakTestDone[1]				:= FALSE;
								bPass[0]						:= FALSE;
								bPass[1]						:= FALSE;
								bFail[0]						:= FALSE;
								bFail[1]						:= FALSE;
								
								IF bError[0] OR bError[1] THEN

									stLeakTesters.State		:= E_LeakTester_State.ERROR;

								ELSIF stLeakTesters.CMD.bAbort OR stLeakTesters.CMD.bEndCycle THEN
									
									stLeakTesters.State			:= E_LeakTester_State.ABORTED;
									
								ELSE stLeakTesters.State			:= E_LeakTester_State.READY;
								
								END_IF
								
								
								
	E_LeakTester_State.STOPPING: 
	
								bStop[0]						:= TRUE;
								bStop[1]						:= TRUE;
								
								IF tonStationStopped.Q THEN
									
									stLeakTesters.State			:= E_LeakTester_State.RESET;
									
								END_IF
	
	E_LeakTester_State.ERROR:
	
								IF NOT bError[0] AND bError[1] THEN
									
									stLeakTesters.State						:= E_LeakTester_State.ABORTED;
									
								END_IF

ELSE stLeakTesters.State := E_LeakTester_State.ABORTED;
	
END_CASE
/////////////////////////////////////////////////////////////////////////////////////STATUS/////////////////////////////////////////////////////////////////////////////////////

stLeakTesters.Status.bBusy	:= 	stLeakTesters.State = E_LeakTester_State.STOPPING OR
								stLeakTesters.State = E_LeakTester_State.HOMING OR
								stLeakTesters.State = E_LeakTester_State.RUN_LEAK_TESTERS OR
								stLeakTesters.State = E_LeakTester_State.WAIT_LEAK_TESTERS;

stLeakTesters.Status.bDone	:= 	stLeakTesters.State = E_LeakTester_State.DONE;

stLeakTesters.Status.bError	:= 	stLeakTesters.State = E_LeakTester_State.ERROR;	

stLeakTesters.Status.bReady	:=	stLeakTesters.State = E_LeakTester_State.READY;

stLeakTesters.Status.bStopped := NOT stLeakTesters.Status.bBusy;
END_ACTION

ACTION b_ACT_IO:


bStopped[0]								:= NOT LeakTester1_IO.sti28General_I_O.bTestActiveLiveData;
bStopped[1]								:= NOT LeakTester2_IO.sti28General_I_O.bTestActiveLiveData;
bError[0]								:= LeakTester1_IO.sti28General_I_O.bMalfunction;
bError[1]								:= LeakTester2_IO.sti28General_I_O.bMalfunction;
bReady[0]								:= LeakTester1_IO.sti28General_I_O.bInstrumentReady;
bReady[1]								:= LeakTester2_IO.sti28General_I_O.bInstrumentReady;
LeakTester1_IO.sti28General_I_O.bReset	:= bReset[0] OR bLeaktester1_Reset;	
LeakTester2_IO.sti28General_I_O.bReset	:= bReset[1] OR bLeaktester2_Reset;	
LeakTester1_IO.sti28General_I_O.bStart	:= bStart[0] OR bLeaktester1_Start;
LeakTester2_IO.sti28General_I_O.bStart	:= bStart[1] OR bLeaktester2_Start;
LeakTester1_IO.sti28General_I_O.bStop	:= bStop[0] OR bLeaktester1_Stop OR stLeakTesters.CMD.bAbort;
LeakTester2_IO.sti28General_I_O.bStop	:= bStop[1] OR bLeaktester2_Stop OR stLeakTesters.CMD.bAbort;



rReset[0](CLK := stLeakTesters.CMD.bReset, Q => bReset[0]);
rReset[1](CLK := stLeakTesters.CMD.bReset, Q => bReset[1]);

fLeakTestDone[0](CLK := LeakTester1_IO.sti28General_I_O.bTestActiveLiveData);
fLeakTestDone[1](CLK := LeakTester2_IO.sti28General_I_O.bTestActiveLiveData);
rPass[0](CLK := LeakTester1_IO.sti28General_I_O.bProgramAccept);
rPass[1](CLK := LeakTester2_IO.sti28General_I_O.bProgramAccept);
rFail[0](CLK := LeakTester1_IO.sti28General_I_O.bProgramReject);
rFail[1](CLK := LeakTester2_IO.sti28General_I_O.bProgramReject);



IF fLeakTestDone[0].Q THEN
	
	bLeakTestDone[0]					:= TRUE;
	
END_IF

IF fLeakTestDone[1].Q THEN
	
	bLeakTestDone[1]					:= TRUE;
	
END_IF

IF rPass[0].Q THEN
	
	bPass[0]							:= TRUE;

END_IF

IF rPass[1].Q THEN
	
	bPass[1]							:= TRUE;

END_IF

IF rFail[0].Q THEN
	
	bFail[0]							:= TRUE;

END_IF

IF rFail[1].Q THEN
	
	bFail[1]							:= TRUE;

END_IF
END_ACTION

ACTION c_ACT_Statistics_Station_1:
stStatisticsHMI[1].sName			:= 'LEAK TESTER 1';
stStatisticsHMI[2].sName			:= 'LEAK TESTER 2';


rGoodStatistics[0]( CLK := stCycleDataNest1.LeakTest_Pass );
rGoodStatistics[1]( CLK := stCycleDataNest2.LeakTest_Pass );
rBadStatistics[0] ( CLK := stCycleDataNest1.LeakTest_Fail );
rBadStatistics[1] ( CLK := stCycleDataNest2.LeakTest_Fail );

IF 	rGoodStatistics[0].Q THEN
	
	stStatisticsHMI[1].nGood		:= stStatisticsHMI[1].nGood + 1;
	stStatisticsHMI[1].nTotalGood	:= stStatisticsHMI[1].nTotalGood + 1;
	
END_IF
								
IF 	rBadStatistics[0].Q THEN
	
	stStatisticsHMI[1].nBad			:= stStatisticsHMI[1].nBad + 1;
	stStatisticsHMI[1].nTotalBad	:= stStatisticsHMI[1].nTotalBad + 1;
	
END_IF

IF stStatisticsHMI[1].bResetGood THEN
	stStatisticsHMI[1].nGood		:= 0;
END_IF

IF stStatisticsHMI[1].bResetBad THEN
	stStatisticsHMI[1].nBad			:= 0;
END_IF


IF 	rGoodStatistics[1].Q THEN
	
	stStatisticsHMI[2].nGood		:= stStatisticsHMI[2].nGood + 1;
	stStatisticsHMI[2].nTotalGood	:= stStatisticsHMI[2].nTotalGood + 1;
	
END_IF
								
IF 	rBadStatistics[1].Q THEN
	
	stStatisticsHMI[2].nBad			:= stStatisticsHMI[2].nBad + 1;
	stStatisticsHMI[2].nTotalBad	:= stStatisticsHMI[2].nTotalBad + 1;
	
END_IF

IF stStatisticsHMI[2].bResetGood THEN
	stStatisticsHMI[2].nGood		:= 0;
END_IF

IF stStatisticsHMI[2].bResetBad THEN
	stStatisticsHMI[2].nBad			:= 0;
END_IF



IF (( stStatisticsHMI[1].nGood + stStatisticsHMI[1].nBad) <> 0) THEN
	
	rEfficency[0]							:= LREAL_TO_FMTSTR(in := (DINT_TO_REAL(stStatisticsHMI[1].nGood) /( DINT_TO_REAL(stStatisticsHMI[1].nGood) + DINT_TO_REAL(stStatisticsHMI[1].nBad))) * 100.0,iPrecision := 2, bRound := TRUE);
	stStatisticsHMI[1].nEfficency		:= CONCAT(STR1 := '%', STR2 := (rEfficency[0]));

ELSE stStatisticsHMI[1].nEfficency		:= CONCAT(STR1 := '%', STR2 := (DINT_TO_STRING(0)));
	
END_IF

IF (( stStatisticsHMI[2].nGood + stStatisticsHMI[2].nBad) <> 0) THEN
	
	rEfficency[1]							:= LREAL_TO_FMTSTR(in := (DINT_TO_REAL(stStatisticsHMI[2].nGood) /( DINT_TO_REAL(stStatisticsHMI[2].nGood) + DINT_TO_REAL(stStatisticsHMI[2].nBad))) * 100.0,iPrecision := 2, bRound := TRUE);
	stStatisticsHMI[2].nEfficency		:= CONCAT(STR1 := '%', STR2 := (rEfficency[1]));

ELSE stStatisticsHMI[2].nEfficency		:= CONCAT(STR1 := '%', STR2 := (DINT_TO_STRING(0)));
	
END_IF
END_ACTION

ACTION d_ACT_Set_Events_Station_1:
//IMMEDIATE FAULTS

stStationEvents[1].aEvents[0].bFault						:= TRUE;
stStationEvents[1].aEvents[0].bEventTimer( IN := (stLeakTesters.State = E_LeakTester_State.RUN_LEAK_TESTERS) OR (stLeakTesters.State = E_LeakTester_State.WAIT_LEAK_TESTERS), PT := stTimers.tStation1TimeOut);
stStationEvents[1].aEvents[0].bEventFlag					:= stStationEvents[1].aEvents[0].bEventTimer.Q;
stStationEvents[1].aEvents[0].bEventText					:= 'Leak tester cycle Timeout';
stStationEvents[1].aEvents[0].sSolution						:= 'Reset System';



//CYCLE STOP REQUEST

stStationEvents[1].aEvents[20].bCycleStopRequest				:= TRUE;
stStationEvents[1].aEvents[20].bEventFlag					:= NOT bReady[0] AND (stLeakTesters.State = E_LeakTester_State.HOMING);// AND (stLeakTesters.State = E_LeakTester_State.HOMING);
stStationEvents[1].aEvents[20].bEventText					:= 'Leak Tester 1 not ready';
stStationEvents[1].aEvents[20].sSolution						:= 'Check Leak tester 1';

stStationEvents[1].aEvents[21].bCycleStopRequest				:= TRUE;
stStationEvents[1].aEvents[21].bEventFlag					:= NOT bReady[1] AND (stLeakTesters.State = E_LeakTester_State.HOMING);// AND (stLeakTesters.State = E_LeakTester_State.HOMING);
stStationEvents[1].aEvents[21].bEventText					:= 'Leak Tester 2 not ready';
stStationEvents[1].aEvents[21].sSolution						:= 'Check Leak tester 2';

//Message
(*
stStationEvents[1].aEvents[3].bMessage						:= TRUE;
stStationEvents[1].aEvents[3].bEventFlag					:= bEventsFlag[3];
stStationEvents[1].aEvents[3].bEventText					:= 'Message 3';
stStationEvents[1].aEvents[3].sSolution						:= '';*)
END_ACTION

END_PROGRAM

// ---- POUs/B_STATIONS/B_3_CAMERA/B_3_1_PRG_Master_Camera.TcPOU
PROGRAM B_3_1_PRG_Master_Camera

VAR
	
	rGoodStatistics						: ARRAY [0..1] OF R_TRIG;
	rBadStatistics						: ARRAY [0..1] OF R_TRIG;
	rEfficency							: ARRAY [0..1] OF STRING(510);
	bEventsFlag							: ARRAY [0..100] OF BOOL;
/////////////////////////////////////////////////////////////////////////////////////I O/////////////////////////////////////////////////////////////////////////////////////	
	bError								: ARRAY [1..4] OF BOOL;
	rReset								: R_TRIG;
	bReset								: BOOL;
	bReady								: BOOL;
	bDone								: ARRAY [1..2] OF BOOL;
	bPass								: ARRAY [1..2] OF BOOL;
	rsPass								: ARRAY [1..2] OF RS;
	bFail								: ARRAY [1..2] OF BOOL;
	bTtigger							: ARRAY [1..4] OF BOOL;
	bTriggerFail						: ARRAY [1..4] OF BOOL;
	bBusy								: ARRAY [1..4] OF BOOL;
	bGeneralBusy						: BOOL;
	bClearBuffer						: BOOL;
	
END_VAR

d_ACT_Set_Events_Station_3();
a_ACT_Ctrl_Station_3();
b_ACT_IO();
c_ACT_Statistics_Station_3();

ACTION a_ACT_Ctrl_Station_3:
/////////////////////////////////////////////////////////////////////////////////////UTILITIES/////////////////////////////////////////////////////////////////////////////////////

/////////////////////////////////////////////////////////////////////////////////////CONDITIONS/////////////////////////////////////////////////////////////////////////////////////

IF bError[1] OR bError[2] OR bError[3] OR bError[4] OR stCamera.CMD.bAbort THEN
	
	stCamera.State						:= E_Camera_State.RESET_CMD;

END_IF

CASE stCamera.State OF
	
	E_Camera_State.ABORTED:
	
								
								
	
								IF  stCamera.CMD.bEnable THEN
									
									stCamera.State						:= E_Camera_State.HOMING;
								
								END_IF
													
	E_Camera_State.HOMING:
	
								IF bReady THEN
									
									stCamera.State						:= E_Camera_State.READY;
									
								END_IF
	
						
	E_Camera_State.READY:
								bClearBuffer							:= TRUE;
							
								IF stCamera.CMD.bExecute THEN
									
									stCamera.State						:= E_Camera_State.TAKING_PICTURE;
									bClearBuffer						:= FALSE;
									
								END_IF
	
	E_Camera_State.TAKING_PICTURE:
								
								bClearBuffer							:= FALSE;
								
								IF stCamera.CMD.CameraCMD.Inspect1 AND stCamera.CMD.CameraCMD.Inspect2 THEN
									
									bTtigger[1]							:= TRUE;
									bTtigger[2]							:= TRUE;
									bTtigger[3]							:= TRUE;
									bTtigger[4]							:= TRUE;
									
									IF bDone[1] AND bDone[2] AND NOT bGeneralBusy  THEN
										
										bTtigger[1]						:= FALSE;
										bTtigger[2]						:= FALSE;
										bTtigger[3]						:= FALSE;
										bTtigger[4]						:= FALSE;
								
										
										stCamera.State					:= E_Camera_State.RESULTS;
										
									END_IF
									
								ELSIF stCamera.CMD.CameraCMD.Inspect1 AND NOT stCamera.CMD.CameraCMD.Inspect2 THEN
									
									bTtigger[1]							:= TRUE;
									bTtigger[2]							:= TRUE;
									
									IF bDone[1] AND NOT bGeneralBusy THEN
										
										bTtigger[1]						:= FALSE;
										bTtigger[2]						:= FALSE;
									
										
										stCamera.State						:= E_Camera_State.RESULTS;
										
									END_IF
								
								ELSIF NOT stCamera.CMD.CameraCMD.Inspect1 AND stCamera.CMD.CameraCMD.Inspect2 THEN
									
									bTtigger[3]							:= TRUE;
									bTtigger[4]							:= TRUE;
									
									IF bDone[2] AND NOT bGeneralBusy THEN

										bTtigger[3]						:= FALSE;
										bTtigger[4]						:= FALSE;
										
										stCamera.State						:= E_Camera_State.RESULTS;
										
									END_IF
								
									
								END_IF
								
								
	E_Camera_State.RESULTS:
								IF stCamera.CMD.CameraCMD.Inspect1 THEN
									
									IF rsPass[1].Q1 THEN
									
										bPass[1]							:= TRUE;
									
									ELSE bFail[1]							:= TRUE;
									
									END_IF
								
								END_IF
								
								IF stCamera.CMD.CameraCMD.Inspect2 THEN
								
									IF rsPass[2].Q1 THEN
									
										bPass[2]							:= TRUE;
									
									ELSE bFail[2]							:= TRUE;
									
									END_IF
								END_IF
								
								stCycleDataNest1.Camera_Pass			:= bPass[1];
								stCycleDataNest1.Camera_Fail			:= bFail[1];
								stCycleDataNest2.Camera_Pass			:= bPass[2];
								stCycleDataNest2.Camera_Fail			:= bFail[2];
								
								Camera1_IO.bResultReadyAck				:= FALSE;
								Camera2_IO.bResultReadyAck				:= FALSE;
								Camera3_IO.bResultReadyAck				:= FALSE;
								Camera4_IO.bResultReadyAck				:= FALSE;
								stCamera.State						:= E_Camera_State.DONE;
								
		E_Camera_State.DONE:		
	
								IF stCamera.CMD.bAcknowledge THEN
									
									stCamera.CMD.bAcknowledge			:= FALSE;
									stCamera.State						:= E_Camera_State.RESET_CMD;
								
								END_IF
								
	E_Camera_State.RESET_CMD:						
	
								
									
								bTtigger[1]								:= FALSE;
								bTtigger[2]								:= FALSE;
								bTtigger[3]								:= FALSE;
								bTtigger[4]								:= FALSE;
								
								bPass[1]								:= FALSE;
								bPass[2]								:= FALSE;
								bFail[1]								:= FALSE;
								bFail[2]								:= FALSE;
								
					
								IF  bError[1] OR bError[2] OR bError[3] OR bError[4] THEN
									
									stCamera.State						:= E_Camera_State.ERROR;
									
								ELSIF  stCamera.CMD.bAbort THEN

									stCamera.State						:= E_Camera_State.ABORTED;
								
								ELSE 
									stCamera.State						:= E_Camera_State.READY;
								END_IF
								
								

								
	
	E_Camera_State.ERROR:	
	
								IF NOT bError[1] OR bError[2] OR bError[3] OR bError[4] THEN
									
									stCamera.State					:= E_Camera_State.ABORTED;
								
								END_IF
					
								
									

ELSE stCamera.State						:= E_Camera_State.READY;
	
END_CASE
/////////////////////////////////////////////////////////////////////////////////////STATUS/////////////////////////////////////////////////////////////////////////////////////

stCamera.Status.bBusy		:= 	stCamera.State	= E_Camera_State.TAKING_PICTURE;
								
stCamera.Status.bDone		:=	stCamera.State	= E_Camera_State.DONE;
											
stCamera.Status.bError		:= 	stCamera.State	= E_Camera_State.ERROR;

stCamera.Status.bReady		:= 	stCamera.State	= E_Camera_State.READY;

stCamera.Status.bStopped	:= 	NOT stCamera.Status.bBusy;
END_ACTION

ACTION b_ACT_IO:

bError[1]								:= Camera1_IO.bError;
bError[2]								:= Camera2_IO.bError;
bError[3]								:= Camera3_IO.bError;
bError[4]								:= Camera4_IO.bError;

bReady									:=  (Camera1_IO.bReady AND Camera1_IO.bRun) AND (Camera2_IO.bReady AND Camera2_IO.bRun) AND 
											(Camera3_IO.bReady AND Camera3_IO.bRun) AND (Camera4_IO.bReady AND Camera4_IO.bRun);

bDone[1]								:= Camera1_IO.bResultReady AND Camera2_IO.bResultReady;
bDone[2]								:= Camera3_IO.bResultReady AND Camera4_IO.bResultReady;

rsPass[1]( SET := bDone[1] AND (Camera1_IO.bTotalResult = TRUE AND Camera2_IO.bTotalResult = TRUE), RESET1 := (stCamera.State = E_Camera_State.ABORTED) OR (stCamera.State = E_Camera_State.READY));
rsPass[2]( SET := bDone[2] AND (Camera3_IO.bTotalResult = TRUE AND Camera4_IO.bTotalResult = TRUE), RESET1 := (stCamera.State = E_Camera_State.ABORTED) OR (stCamera.State = E_Camera_State.READY));


bBusy[1]								:= Camera1_IO.bBusy;
bBusy[2]								:= Camera2_IO.bBusy;
bBusy[3]								:= Camera3_IO.bBusy;
bBusy[4]								:= Camera4_IO.bBusy;

bGeneralBusy							:= bBusy[1] OR bBusy[2] OR bBusy[3] OR bBusy[4];

bTriggerFail[1]							:= Camera1_IO.bTriggerFail;
bTriggerFail[2]							:= Camera2_IO.bTriggerFail;
bTriggerFail[3]							:= Camera3_IO.bTriggerFail;
bTriggerFail[4]							:= Camera4_IO.bTriggerFail;

Camera1_IO.bReset						:= bReset;
Camera2_IO.bReset						:= bReset;
Camera3_IO.bReset						:= bReset;
Camera4_IO.bReset						:= bReset;

Camera1_IO.bTrigger						:= bTtigger[1] OR bCameraTrigger[1];	
Camera2_IO.bTrigger						:= bTtigger[2] OR bCameraTrigger[2];
Camera3_IO.bTrigger						:= bTtigger[3] OR bCameraTrigger[3];
Camera4_IO.bTrigger						:= bTtigger[4] OR bCameraTrigger[4];

IF bClearBuffer	THEN
	
	Camera1_IO.bClearBuffer				:= TRUE;
	Camera2_IO.bClearBuffer				:= TRUE;
	Camera3_IO.bClearBuffer				:= TRUE;
	Camera4_IO.bClearBuffer				:= TRUE;

ELSE

	Camera1_IO.bClearBuffer				:= FALSE;
	Camera2_IO.bClearBuffer				:= FALSE;
	Camera3_IO.bClearBuffer				:= FALSE;
	Camera4_IO.bClearBuffer				:= FALSE;

END_IF

//////////////////////////////////////////////////////////////////////HMI//////////////////////////////////////////////////////////////////////////////
bCameraSettingNo[1]						:= 2;
bCameraSettingNo[2]						:= 2;
bCameraSettingNo[3]						:= 2;
bCameraSettingNo[4]						:= 2;


Camera1_IO.bResetStatistics				:= bCameraResetStatistics[1];
Camera1_IO.bSettingNo					:= bCameraSettingNo[1];
Camera1_IO.bSettingVal					:= bCameraSettingVal[1];
Camera1_IO.bSetTreshold					:= bCameraSetTreshold[1];

Camera2_IO.bResetStatistics				:= bCameraResetStatistics[2];
Camera2_IO.bSettingNo					:= bCameraSettingNo[2];
Camera2_IO.bSettingVal					:= bCameraSettingVal[2];
Camera2_IO.bSetTreshold					:= bCameraSetTreshold[2];

Camera3_IO.bResetStatistics				:= bCameraResetStatistics[3];
Camera3_IO.bSettingNo					:= bCameraSettingNo[3];
Camera3_IO.bSettingVal					:= bCameraSettingVal[3];
Camera3_IO.bSetTreshold					:= bCameraSetTreshold[3];

Camera4_IO.bResetStatistics				:= bCameraResetStatistics[4];
Camera4_IO.bSettingNo					:= bCameraSettingNo[4];
Camera4_IO.bSettingVal					:= bCameraSettingVal[4];
Camera4_IO.bSetTreshold					:= bCameraSetTreshold[4];

//Camera1_IO.bTriggerFail

rReset( CLK := stCamera.CMD.bReset, Q => bReset);
END_ACTION

ACTION c_ACT_Statistics_Station_3:
stStatisticsHMI[5].sName			:= 'Vision System 1';
stStatisticsHMI[6].sName			:= 'Vision System 2';


rGoodStatistics[0]( CLK := stCycleDataNest1.Camera_Pass);
rBadStatistics[0]( CLK := stCycleDataNest1.Camera_Fail);
rGoodStatistics[1]( CLK := stCycleDataNest2.Camera_Pass);
rBadStatistics[1]( CLK := stCycleDataNest2.Camera_Fail);

IF 	rGoodStatistics[0].Q THEN
	
	stStatisticsHMI[5].nGood		:= stStatisticsHMI[5].nGood + 1;
	stStatisticsHMI[5].nTotalGood	:= stStatisticsHMI[5].nTotalGood + 1;
	
END_IF
								
IF 	rBadStatistics[0].Q THEN
	
	stStatisticsHMI[5].nBad			:= stStatisticsHMI[5].nBad + 1;
	stStatisticsHMI[5].nTotalBad	:= stStatisticsHMI[5].nTotalBad + 1;
	
END_IF

IF stStatisticsHMI[5].bResetGood THEN
	stStatisticsHMI[5].nGood		:= 0;
END_IF

IF stStatisticsHMI[5].bResetBad THEN
	stStatisticsHMI[5].nBad			:= 0;
END_IF

IF 	rGoodStatistics[1].Q THEN
	
	stStatisticsHMI[6].nGood		:= stStatisticsHMI[6].nGood + 1;
	stStatisticsHMI[6].nTotalGood	:= stStatisticsHMI[6].nTotalGood + 1;
	
END_IF
								
IF 	rBadStatistics[1].Q THEN
	
	stStatisticsHMI[6].nBad			:= stStatisticsHMI[6].nBad + 1;
	stStatisticsHMI[6].nTotalBad	:= stStatisticsHMI[6].nTotalBad + 1;
	
END_IF

IF stStatisticsHMI[6].bResetGood THEN
	stStatisticsHMI[6].nGood		:= 0;
END_IF

IF stStatisticsHMI[6].bResetBad THEN
	stStatisticsHMI[6].nBad			:= 0;
END_IF

IF (( stStatisticsHMI[5].nGood + stStatisticsHMI[5].nBad) <> 0) THEN
	
	rEfficency[0]							:= LREAL_TO_FMTSTR(in := (DINT_TO_REAL(stStatisticsHMI[5].nGood) /( DINT_TO_REAL(stStatisticsHMI[5].nGood) + DINT_TO_REAL(stStatisticsHMI[5].nBad))) * 100.0,iPrecision := 2, bRound := TRUE);
	stStatisticsHMI[5].nEfficency		:= CONCAT(STR1 := '%', STR2 := (rEfficency[0]));

ELSE stStatisticsHMI[5].nEfficency		:= CONCAT(STR1 := '%', STR2 := (DINT_TO_STRING(0)));
	
END_IF

IF (( stStatisticsHMI[6].nGood + stStatisticsHMI[6].nBad) <> 0) THEN
	
	rEfficency[1]							:= LREAL_TO_FMTSTR(in := (DINT_TO_REAL(stStatisticsHMI[6].nGood) /( DINT_TO_REAL(stStatisticsHMI[6].nGood) + DINT_TO_REAL(stStatisticsHMI[6].nBad))) * 100.0,iPrecision := 2, bRound := TRUE);
	stStatisticsHMI[6].nEfficency		:= CONCAT(STR1 := '%', STR2 := (rEfficency[1]));

ELSE stStatisticsHMI[6].nEfficency		:= CONCAT(STR1 := '%', STR2 := (DINT_TO_STRING(0)));
	
END_IF
END_ACTION

ACTION d_ACT_Set_Events_Station_3:
//IMMEDIATE FAULTS

stStationEvents[3].aEvents[0].bFault						:= TRUE;
stStationEvents[3].aEvents[0].bEventFlag					:= bError[1];
stStationEvents[3].aEvents[0].bEventText					:= 'Error camera 1';
stStationEvents[3].aEvents[0].sSolution						:= 'Check camera 1';

stStationEvents[3].aEvents[1].bFault						:= TRUE;
stStationEvents[3].aEvents[1].bEventFlag					:= bError[2];
stStationEvents[3].aEvents[1].bEventText					:= 'Error camera 2';
stStationEvents[3].aEvents[1].sSolution						:= 'Check camera 2';

stStationEvents[3].aEvents[2].bFault						:= TRUE;
stStationEvents[3].aEvents[2].bEventFlag					:= bError[3];
stStationEvents[3].aEvents[2].bEventText					:= 'Error camera 3';
stStationEvents[3].aEvents[2].sSolution						:= 'Check camera 3';

stStationEvents[3].aEvents[3].bFault						:= TRUE;
stStationEvents[3].aEvents[3].bEventFlag					:= bError[4];
stStationEvents[3].aEvents[3].bEventText					:= 'Error camera 4';
stStationEvents[3].aEvents[3].sSolution						:= 'Check camera 4';

stStationEvents[3].aEvents[4].bFault						:= TRUE;
stStationEvents[3].aEvents[4].bEventTimer(IN := stCamera.Status.bBusy, PT := stTimers.tStation3TimeOut);
stStationEvents[3].aEvents[4].bEventFlag					:= stStationEvents[3].aEvents[4].bEventTimer.Q;
stStationEvents[3].aEvents[4].bEventText					:= 'Camera Cycle Timeout';
stStationEvents[3].aEvents[4].sSolution						:= 'Reset Sytem';


//CYCLE STOP FAULT

stStationEvents[3].aEvents[20].bCycleStopRequest			:= TRUE;
stStationEvents[3].aEvents[20].bEventFlag					:= bTriggerFail[1];
stStationEvents[3].aEvents[20].bEventText					:= 'Trigger failed in camera 1';
stStationEvents[3].aEvents[20].sSolution					:= 'Check camera 1';

stStationEvents[3].aEvents[21].bCycleStopRequest			:= TRUE;
stStationEvents[3].aEvents[21].bEventFlag					:= bTriggerFail[2];
stStationEvents[3].aEvents[21].bEventText					:= 'Trigger failed in camera 2';
stStationEvents[3].aEvents[21].sSolution					:= 'Check camera 2';

stStationEvents[3].aEvents[22].bCycleStopRequest			:= TRUE;
stStationEvents[3].aEvents[22].bEventFlag					:= bTriggerFail[3];
stStationEvents[3].aEvents[22].bEventText					:= 'Trigger failed in camera 3';
stStationEvents[3].aEvents[22].sSolution					:= 'Check camera 3';

stStationEvents[3].aEvents[23].bCycleStopRequest			:= TRUE;
stStationEvents[3].aEvents[23].bEventFlag					:= bTriggerFail[4];
stStationEvents[3].aEvents[23].bEventText					:= 'Trigger failed in camera 4';
stStationEvents[3].aEvents[23].sSolution					:= 'Check camera 4';


//CYCLE STOP REQUEST

stStationEvents[3].aEvents[2].bCycleStopRequest				:= TRUE;
stStationEvents[3].aEvents[2].bEventFlag					:= bEventsFlag[2];
stStationEvents[3].aEvents[2].bEventText					:= 'ST1 EVENT 7';
END_ACTION

END_PROGRAM

// ---- POUs/B_STATIONS/B_4_PROCESS_CYLINDER__SLICE_DOOR/B_4_1_PRG_Master_ProcessCylinder.TcPOU
PROGRAM B_4_1_PRG_Master_ProcessCylinder

VAR

	
	
/////////////////////////////////////////////////////////////////////////////////////I O/////////////////////////////////////////////////////////////////////////////////////	
	bExtended							: BOOL;
	bRetracted							: BOOL;
	bExtend								: BOOL;
	bRetract							: BOOL;

	
END_VAR

d_ACT_Set_Events_Station_4A();
a_ACT_Ctrl_Station_4A();
b_ACT_IO_A();
c_Manual();

ACTION a_ACT_Ctrl_Station_4A:
/////////////////////////////////////////////////////////////////////////////////////UTILITIES/////////////////////////////////////////////////////////////////////////////////////

/////////////////////////////////////////////////////////////////////////////////////CONDITIONS/////////////////////////////////////////////////////////////////////////////////////


IF stProcessCylinder.CMD.bAbort THEN
	
	stProcessCylinder.State				:= E_ProcessCylinder_State.RESET;

END_IF

CASE stProcessCylinder.State OF
	
	E_ProcessCylinder_State.ABORTED:
	
								IF stProcessCylinder.CMD.bEnable THEN
									
									stProcessCylinder.State				:= E_ProcessCylinder_State.HOMING;
								
								END_IF
								
	E_ProcessCylinder_State.HOMING:
	
								bRetract								:= TRUE;
								
								IF bRetracted THEN
									
									bRetract							:= FALSE;
									stProcessCylinder.State				:= E_ProcessCylinder_State.READY;
									
								
								END_IF
	
	E_ProcessCylinder_State.READY:
	
								IF stProcessCylinder.CMD.bExecute AND stProcessCylinder.CMD.ProcessCylinderCMD.ExtendCylinder1 THEN

									stProcessCylinder.State				:= E_ProcessCylinder_State.EXTEND;
									
								ELSIF stProcessCylinder.CMD.bExecute AND stProcessCylinder.CMD.ProcessCylinderCMD.RetractCylinder1 THEN
									
									stProcessCylinder.State				:= E_ProcessCylinder_State.RETRACT;;									
																		
								END_IF
	
	E_ProcessCylinder_State.EXTEND:
	
								bExtend									:= stProcessCylinder.CMD.ProcessCylinderCMD.ExtendCylinder1;
								
								IF bExtend THEN
									
									IF bExtended THEN

										stProcessCylinder.State			:= E_ProcessCylinder_State.DONE;
									
									END_IF						
	
								END_IF
								
	E_ProcessCylinder_State.RETRACT:
	
								bRetract								:= stProcessCylinder.CMD.ProcessCylinderCMD.RetractCylinder1;
								
								
								IF bRetract THEN
									
									IF bRetracted THEN

										stProcessCylinder.State				:= E_ProcessCylinder_State.DONE;
									
									END_IF					
	
								END_IF
								
	E_ProcessCylinder_State.DONE:
	
								IF stProcessCylinder.CMD.bAcknowledge THEN
									
									stProcessCylinder.CMD.bAcknowledge		:= FALSE;
									stProcessCylinder.State					:= E_ProcessCylinder_State.RESET;
								
								END_IF
	
	
	E_ProcessCylinder_State.RESET:	
	
								bExtend										:= FALSE;								
								bRetract									:= FALSE;
								
								
								IF NOT stProcessCylinder.CMD.bAbort AND NOT stProcessCylinder.CMD.bEndCycle THEN
									
									stProcessCylinder.State					:= E_ProcessCylinder_State.READY;
									
								ELSE stProcessCylinder.State					:= E_ProcessCylinder_State.ABORTED;
								END_IF
									

ELSE stProcessCylinder.State	:= E_ProcessCylinder_State.ABORTED;
	
END_CASE
/////////////////////////////////////////////////////////////////////////////////////STATUS/////////////////////////////////////////////////////////////////////////////////////

stProcessCylinder.Status.bBusy		:= 	stProcessCylinder.State	= E_ProcessCylinder_State.EXTEND OR
										stProcessCylinder.State	= E_ProcessCylinder_State.RETRACT OR 
										stProcessCylinder.State	= E_ProcessCylinder_State.STOPPING;
								
stProcessCylinder.Status.bDone		:=	stProcessCylinder.State	= E_ProcessCylinder_State.DONE;

stProcessCylinder.Status.bReady		:= 	stProcessCylinder.State	= E_ProcessCylinder_State.READY;

stProcessCylinder.Status.bStopped	:= 	NOT stProcessCylinder.Status.bBusy;
END_ACTION

ACTION b_ACT_IO_A:

bExtended								:= dw_T08_EL1809.iProcessCylinder1Extended;
bRetracted								:= stTwinSAFE.qProcessCylinder1Retracted;

dw_T09_EL2809.qExtendProcessCylinder1	:= bExtend OR bProcessCylinder1_Down ;	
dw_T09_EL2809.qRetractProcessCylinder1	:= bRetract OR bProcessCylinder1_Up OR bProcessCylinderSafetyPosition;

IF stStationEvents[3].aEvents[0].bEventTimer.Q THEN
	
	bRetract := FALSE;

END_IF

IF stStationEvents[3].aEvents[1].bEventTimer.Q THEN
	
	bExtended := FALSE;

END_IF
END_ACTION

ACTION c_Manual:
(*
IF bProcessCylinder1_Up THEN
	
	bRetract[0] := TRUE;
	
ELSIF bRetracted[0] THEN
	
	bRetract[0] := FALSE;

END_IF

IF bProcessCylinder1_Down THEN
	
	bExtend[0] := TRUE;
	
ELSIF bExtended[0] THEN
	
	bExtend[0] := FALSE;

END_IF

IF bProcessCylinder2_Up THEN
	
	bRetract[1] := TRUE;
	
ELSIF bRetracted[1] THEN
	
	bRetract[1] := FALSE;

END_IF

IF bProcessCylinder2_Down THEN
	
	bExtend[1] := TRUE;
	
ELSIF bExtended[1] THEN
	
	bExtend[1] := FALSE;

END_IF
*)
END_ACTION

ACTION d_ACT_Set_Events_Station_4A:
//FAULTS

stStationEvents[3].aEvents[0].bEventTimer( IN := (bExtend AND NOT bExtended), PT := T#5S);
stStationEvents[3].aEvents[0].bFault						:= TRUE;
stStationEvents[3].aEvents[0].bEventFlag					:= stStationEvents[3].aEvents[0].bEventTimer.Q;
stStationEvents[3].aEvents[0].bEventText					:= 'Process Cylinder 1 extend timeout';
stStationEvents[3].aEvents[0].sSolution						:= 'Check cylinder, neumatic connections and sensors';

stStationEvents[3].aEvents[1].bEventTimer( IN := (bRetract AND NOT bRetracted), PT := T#5S);
stStationEvents[3].aEvents[1].bFault						:= TRUE;
stStationEvents[3].aEvents[1].bEventFlag					:= stStationEvents[3].aEvents[1].bEventTimer.Q;
stStationEvents[3].aEvents[1].bEventText					:= 'Process Cylinder retract timeout';
stStationEvents[3].aEvents[1].sSolution						:= 'Check cylinder, neumatic connections and sensors';


//CYCLE STOP REQUEST

(*stStationEvents[3].aEvents[2].bCycleStopRequest			:= TRUE;
stStationEvents[3].aEvents[2].bEventFlag					:= ;
stStationEvents[3].aEvents[2].bEventText					:= 'ST1 EVENT 7';*)
END_ACTION

END_PROGRAM

// ---- POUs/B_STATIONS/B_4_PROCESS_CYLINDER__SLICE_DOOR/B_4_2_PRG_Master_ProcessDoor.TcPOU
PROGRAM B_4_2_PRG_Master_ProcessDoor

VAR

	bEventsFlag							: ARRAY [0..100] OF BOOL;
/////////////////////////////////////////////////////////////////////////////////////I O/////////////////////////////////////////////////////////////////////////////////////	
	
	bOpenDoor							: BOOL;
	bCloseDoor							: BOOL;
	bCloseDoorHMI						: BOOL;
	bDoorClosed							: BOOL;
	tonDoorOpened						: TON;
	bDoorOpened							: BOOL;
	
	
END_VAR

d_ACT_Set_Events_Station_4B();
a_ACT_Ctrl_Station_4B();
b_ACT_IO_B();
c_Manual();

ACTION a_ACT_Ctrl_Station_4B:
/////////////////////////////////////////////////////////////////////////////////////UTILITIES/////////////////////////////////////////////////////////////////////////////////////

/////////////////////////////////////////////////////////////////////////////////////CONDITIONS/////////////////////////////////////////////////////////////////////////////////////


IF stProcessDoor.CMD.bAbort THEN
	
	stProcessDoor.State				:= E_ProcessDoor_State.RESET;
	
ELSIF stProcessDoor.CMD.bEndCycle THEN
	
	stProcessDoor.State				:= E_ProcessDoor_State.STOPPING;

END_IF

CASE stProcessDoor.State OF
	
	E_ProcessDoor_State.ABORTED:
	
								IF stProcessDoor.CMD.bEnable THEN
									
									stProcessDoor.State				:= E_ProcessDoor_State.HOMING;
								
								END_IF
								
		E_ProcessDoor_State.HOMING: 
	
								bOpenDoor							:= TRUE;
								
								IF bDoorOpened THEN
									
									stProcessDoor.State				:= E_ProcessDoor_State.READY;									
									bOpenDoor						:= FALSE;
																	
								END_IF
	
	
	E_ProcessDoor_State.READY:
	
								IF stProcessDoor.CMD.bExecute AND 	stProcessDoor.CMD.ProcessDoorCMD.OpenDoor	THEN

									stProcessDoor.State				:= E_ProcessDoor_State.OPEN;
									
								ELSIF stProcessDoor.CMD.bExecute AND 	stProcessDoor.CMD.ProcessDoorCMD.CloseDoor	THEN
									
									stProcessDoor.State				:= E_ProcessDoor_State.CLOSE;									
																		
								END_IF
	

	E_ProcessDoor_State.OPEN:
	
								bOpenDoor							:= TRUE;
								
								IF bDoorOpened	THEN
									
									stProcessDoor.State				:= E_ProcessDoor_State.DONE;
								
								END_IF
								
	E_ProcessDoor_State.CLOSE:
	
								bCloseDoor							:= TRUE;
								
								IF bDoorClosed THEN
									
									stProcessDoor.State				:= E_ProcessDoor_State.DONE;
								
								END_IF
								
	E_ProcessDoor_State.DONE:
	
	
								IF stProcessDoor.CMD.bAcknowledge THEN
									
									stProcessDoor.CMD.bAcknowledge	:= FALSE;
									stProcessDoor.State				:= E_ProcessDoor_State.RESET;
								
								END_IF
	
	
	E_ProcessDoor_State.RESET:	
	
								bOpenDoor							:= FALSE;
								bCloseDoor							:= FALSE;
								
								IF NOT stProcessDoor.CMD.bAbort AND NOT stProcessDoor.CMD.bEndCycle THEN
									
									stProcessDoor.State				:= E_ProcessDoor_State.READY;
									
								ELSE stProcessDoor.State			:= E_ProcessDoor_State.ABORTED;
								END_IF
	
					
	E_ProcessDoor_State.STOPPING:					
									
								bOpenDoor							:= TRUE;
									
								IF bDoorOpened THEN
									
									bOpenDoor						:= FALSE;
									stProcessDoor.State				:= E_ProcessDoor_State.RESET;
								
								END_IF
								
							
														
									

ELSE stProcessDoor.State		:= E_ProcessDoor_State.ABORTED;
	
END_CASE
/////////////////////////////////////////////////////////////////////////////////////STATUS/////////////////////////////////////////////////////////////////////////////////////

stProcessDoor.Status.bBusy			:= 	stProcessDoor.State	= E_ProcessDoor_State.CLOSE OR
										stProcessDoor.State	= E_ProcessDoor_State.OPEN OR 
										stProcessDoor.State	= E_ProcessDoor_State.STOPPING;
								
stProcessDoor.Status.bDone			:=	stProcessDoor.State	= E_ProcessDoor_State.DONE;

stProcessDoor.Status.bReady			:= 	stProcessDoor.State	= E_ProcessDoor_State.READY;

stProcessDoor.Status.bStopped		:= 	NOT stProcessDoor.Status.bBusy;
END_ACTION

ACTION b_ACT_IO_B:
tonDoorOpened( IN := NOT bDoorClosed, PT := stTimers.tDoorOpenedSignal);


bDoorClosed								:= dw_T05_EL1918.iProcessDoorClosed1 AND dw_T05_EL1918.iProcessDoorClosed2 AND dw_T05_EL1918.iProcessDoorFB;
bDoorOpened								:= tonDoorOpened.Q; 


dw_T09_EL2809.qOpenProcessDoor	:= bOpenDoor OR bProcessDoor_Up OR bProcessDoorUpInitialising;	
dw_T09_EL2809.qCloseProcessDoor	:= bCloseDoor OR bCloseDoorHMI;
END_ACTION

ACTION c_Manual:

IF bProcessDoor_Down AND dw_T05_EL1918.iLeftTouchButtonNO AND dw_T05_EL1918.iRightTouchButtonNO THEN
	
	bCloseDoorHMI					:= TRUE;
	bProcessDoor_Down				:= FALSE;
	
ELSE bCloseDoorHMI					:= FALSE;

END_IF
END_ACTION

ACTION d_ACT_Set_Events_Station_4B:
//IMMEDIATE FAULTS

stStationEvents[4].aEvents[0].bEventTimer( IN := bCloseDoor AND NOT bDoorClosed, PT := T#5S);
stStationEvents[4].aEvents[0].bFault						:= TRUE;
stStationEvents[4].aEvents[0].bEventFlag					:= stStationEvents[4].aEvents[0].bEventTimer.Q;
stStationEvents[4].aEvents[0].bEventText					:= 'Process Door extend timeout';
stStationEvents[4].aEvents[0].sSolution						:= 'Check cylinder, neumatic connections and sensors';

stStationEvents[4].aEvents[1].bEventTimer( IN := bOpenDoor AND NOT bDoorOpened, PT := T#5S);
stStationEvents[4].aEvents[1].bFault						:= TRUE;
stStationEvents[4].aEvents[1].bEventFlag					:= stStationEvents[4].aEvents[1].bEventTimer.Q;
stStationEvents[4].aEvents[1].bEventText					:= 'Process Door Retract timeout';
stStationEvents[4].aEvents[1].sSolution						:= 'Check cylinder, neumatic connections and sensors';





//CYCLE STOP REQUEST

(*stStationEvents[4].aEvents[2].bCycleStopRequest			:= TRUE;
stStationEvents[4].aEvents[2].bEventFlag					:= bEventsFlag[2];
stStationEvents[4].aEvents[2].bEventText					:= 'ST1 EVENT 7';*)
END_ACTION

END_PROGRAM

// ---- POUs/A_MASTER/A_2_PRG_MachineCtrl.TcPOU
PROGRAM A_2_PRG_MachineCtrl
VAR
/////////////////////////////////////////////////////////////////////////////////////TIMERS & TRIGGERS/////////////////////////////////////////////////////////////////////////////////////

	tonSys_Init					: Tc2_Standard.TON:=(PT:=T#1S);
	tonSys_InitTimeout			: Tc2_Standard.TON:=(PT:=T#20S);					
	tonFirstAutoCycle			: Tc2_Standard.TON:=(PT:=T#500MS);
	
/////////////////////////////////////////////////////////////////////////////////////PROCESS CYCLE/////////////////////////////////////////////////////////////////////////////////////	
	
	eCycleState					: E_General_ProcessCycle;
	tonCMD_Done					: TON;
	tonResetAllCMD				: TON;
	tonExecute					: TON;
	tonSave_Data				: TON;
	tonWriteToCsv				: TON;
	rFirstAutoCycle				: R_TRIG;
	
	bStartProcessCondition		: BOOL;
	i							: INT;
	j							: INT;
	
	abLeakTesterFlag			: ARRAY[0..1] OF BOOL;
	abHeightTestFlag			: ARRAY[0..1] OF BOOL;
	bVisionProcessDoneFlag		: BOOL;
	tonGettingResults			: TON;
	tonWaitExtendCylidner		: TON;

	

/////////////////////////////////////////////////////////////////////////////////////I/O/////////////////////////////////////////////////////////////////////////////////////	

	bPartPresentNest1			: BOOL;
	bPartPresentNest2			: BOOL;
	bPartPresentNest3			: BOOL;
	bPartPresentNest4			: BOOL;
	bRejectSensor				: BOOL;
	bTwoHandsSignal				: BOOL;
	tonTwoHandsSignal			: TON;
	
	bEndAutoCycleFlag			: BOOL;
	bProcessedPart				: ARRAY[0..1] OF BOOL;
	fProcessedPart				: ARRAY[0..1] OF F_TRIG;
	
	
END_VAR

/////////////////////////////////////////////////////////////////////////////////////GENERAL/////////////////////////////////////////////////////////////////////////////////////
a_ACT_MachineStatus();
b_ACT_ProcessCycle();
d_ACT_IO();

ACTION a_ACT_MachineStatus:
/////////////////////////////////////////////////////////////////////////////////////Utilities/////////////////////////////////////////////////////////////////////////////////////
tonSys_Init(IN:=stMachineStatus.bInitialising);
tonSys_InitTimeout(IN:=stMachineStatus.bInitialising);
tonSafety( IN := stMachineStatus.eMachineState = E_MachineState.SAFETY, PT := T#10S);
	
	IF stMachineStatus.eMachineState <> E_MachineState.SYSTEM_AUTO_CYCLE THEN
		
		sMachineMessage									:= '';			
		
	END_IF
/////////////////////////////////////////////////////////////////////////////////////CONDITIONS/////////////////////////////////////////////////////////////////////////////////////
				IF NOT stMasterCtrl.bNoFault THEN
					stMachineStatus.eMachineState 		:= E_MachineState.FAULT;
				END_IF
				
				IF stMachineStatus.eMachineState		= E_MachineState.STOPPING OR
				stMachineStatus.eMachineState			= E_MachineState.FAULT THEN
					
					stCamera.CMD.bAbort					:= TRUE;	
					stLeakTesters.CMD.bAbort			:= TRUE;	
					stHeightTests.CMD.bAbort			:= TRUE;
					stProcessCylinder.CMD.bAbort		:= TRUE;
					stProcessDoor.CMD.bAbort			:= TRUE;
				
					stCamera.CMD.bEnable				:= FALSE;	
					stLeakTesters.CMD.bEnable			:= FALSE;	
					stHeightTests.CMD.bEnable			:= FALSE;
					stProcessCylinder.CMD.bEnable		:= FALSE;
					stProcessDoor.CMD.bEnable			:= FALSE;
					
				END_IF
				
				IF 	stButtonsLamps.bResetButtonFallingEdge THEN
					stCamera.CMD.bReset					:= TRUE;	
					stLeakTesters.CMD.bReset			:= TRUE;	
					stHeightTests.CMD.bReset			:= TRUE;
					stProcessCylinder.CMD.bReset		:= TRUE;
					stProcessDoor.CMD.bReset			:= TRUE;
				ELSE 
					stCamera.CMD.bReset					:= FALSE;	
					stLeakTesters.CMD.bReset			:= FALSE;	
					stHeightTests.CMD.bReset			:= FALSE;
					stProcessCylinder.CMD.bReset		:= FALSE;
					stProcessDoor.CMD.bReset			:= FALSE;
				END_IF	

				IF 	NOT (stMachineStatus.eMachineState = E_MachineState.MANUAL_MODE) THEN
					
					stCamera.CMD.bManualMode				:=FALSE;
					stLeakTesters.CMD.bManualMode			:=FALSE;
					stHeightTests.CMD.bManualMode			:=FALSE;
					stProcessCylinder.CMD.bManualMode		:=FALSE;
					stProcessDoor.CMD.bManualMode			:=FALSE;
					
				END_IF
				
/////////////////////////////////////////////////////////////////////////////////////MACHINE CONTROL/////////////////////////////////////////////////////////////////////////////////////

CASE stMachineStatus.eMachineState OF

E_MachineState.SYSTEM_POWER_UP: 		

				IF tonSystemPowerUP.Q THEN
						stMachineStatus.eMachineState 	:= E_MachineState.STOPPED;//
				END_IF
	
E_MachineState.STOPPED:		

				IF stMasterCtrl.bNoFault   AND NOT stMasterCtrl.bCycleStopRequest AND dw_T04_EL1918.iResetButton THEN
						stMachineStatus.eMachineState 	:= E_MachineState.SAFETY;//
				ELSIF NOT stMasterCtrl.bNoFault    THEN	
					stMachineStatus.eMachineState 		:= E_MachineState.FAULT;		
				END_IF	

E_MachineState.SAFETY:


					IF stTwinSAFE.qSafetyOk AND tonSafety.Q THEN
						
						stMachineStatus.eMachineState 	:= E_MachineState.SYSTEM_INITIALISING;
						
					ELSIF stMasterCtrl.bCycleStopRequest AND stMasterCtrl.bNoFault THEN

						stMachineStatus.eMachineState 	:= E_MachineState.STOPPING;
						
					ELSIF NOT stMasterCtrl.bNoFault THEN
						
						stMachineStatus.eMachineState 		:= E_MachineState.FAULT;	
						
					END_IF

E_MachineState.SYSTEM_INITIALISING:		
					
					
				stCamera.CMD.bAbort						:= FALSE;	
				stLeakTesters.CMD.bAbort				:= FALSE;	
				stHeightTests.CMD.bAbort				:= FALSE;
				stProcessCylinder.CMD.bAbort			:= FALSE;
				stProcessDoor.CMD.bAbort				:= FALSE;	

				IF tonSys_Init.Q THEN
					stCamera.CMD.bEnable				:= TRUE;	
					stLeakTesters.CMD.bEnable			:= TRUE;	
					stHeightTests.CMD.bEnable			:= TRUE;
					stProcessCylinder.CMD.bEnable		:= TRUE;
					stProcessDoor.CMD.bEnable			:= TRUE;						
				END_IF
				
				IF stMasterCtrl.bAllStationsReady  THEN 
					stMachineStatus.eMachineState		:= E_MachineState.SYSTEM_READY_TO_START;
				ELSIF stButtonsLamps.bStopButtonFallingEdge OR  
				stMasterCtrl.bCycleStopRequest OR tonSys_InitTimeout.Q  THEN
					stMachineStatus.eMachineState 		:= E_MachineState.STOPPING;	
				ELSIF NOT stMasterCtrl.bNoFault THEN		
					stMachineStatus.eMachineState 		:= E_MachineState.FAULT;
				END_IF
			
					
E_MachineState.SYSTEM_READY_TO_START:	

				IF 	 stButtonsLamps.bStartButtonFallingEdge AND stMasterCtrl.bAllStationsReady  THEN
					stMachineStatus.eMachineState 		:= E_MachineState.SYSTEM_AUTO_CYCLE;
				ELSIF NOT stMasterCtrl.bAllStationsReady OR stMasterCtrl.bCycleStopRequest THEN
					stMachineStatus.eMachineState 		:= E_MachineState.STOPPING;		
				ELSIF NOT stMasterCtrl.bNoFault THEN	
					stMachineStatus.eMachineState 		:= E_MachineState.FAULT;
				ELSIF GVL_Master.stMasterCTRL.bManualModeRequest AND stMasterCtrl.bNoFault AND bHMIInitialized  THEN
					stMachineStatus.eMachineState 		:= E_MachineState.MANUAL_MODE;
				END_IF

				

E_MachineState.SYSTEM_AUTO_CYCLE:		

				
				IF  stMasterCtrl.bCycleStopRequest AND (eCycleState = E_General_ProcessCycle.IDLE) THEN
	
					stMachineStatus.eMachineState 		:= E_MachineState.STOPPING;
				
				ELSIF stMasterCtrl.bCycleStopRequest AND NOT (eCycleState = E_General_ProcessCycle.IDLE) THEN					
				
					sMachineMessage						:= 'Ending  Cycle';
				
				ELSIF NOT stMasterCtrl.bNoFault THEN	
					stMachineStatus.eMachineState 		:= E_MachineState.FAULT;
				END_IF
				

E_MachineState.STOPPING:	

				
				IF stMasterCtrl.bAllStationsStopped THEN
					stMachineStatus.eMachineState 		:= E_MachineState.STOPPED;
				ELSIF NOT stMasterCtrl.bNoFault THEN	
					stMachineStatus.eMachineState 		:= E_MachineState.FAULT;					
				END_IF
				

E_MachineState.FAULT:	
				
				IF stMasterCtrl.bNoFault	THEN
					stMachineStatus.eMachineState		:= E_MachineState.STOPPED;		
				END_IF

E_MachineState.MANUAL_MODE:

				IF stButtonsLamps.bStopButtonFallingEdge OR NOT GVL_Master.stMasterCTRL.bManualModeRequest THEN
					stMachineStatus.eMachineState 		:= E_MachineState.STOPPING;
				ELSIF  NOT stMasterCtrl.bNoFault THEN	
					stMachineStatus.eMachineState 		:= E_MachineState.FAULT;								
				ELSE 
					
					stCamera.CMD.bManualMode				:=TRUE;
					stLeakTesters.CMD.bManualMode			:=TRUE;
					stHeightTests.CMD.bManualMode			:=TRUE;
					stProcessCylinder.CMD.bManualMode		:=TRUE;
					stProcessDoor.CMD.bManualMode			:=TRUE;

				END_IF
ELSE
stMachineStatus.eMachineState:=E_MachineState.SYSTEM_POWER_UP;		
END_CASE									


/////////////////////////////////////////////////////////////////////////////////////MACHINE STATUS/////////////////////////////////////////////////////////////////////////////////////
stMachineStatus.bSystemPowerUp 			:= (stMachineStatus.eMachineState = E_MachineState.SYSTEM_POWER_UP);
stMachineStatus.bStopped 				:= (stMachineStatus.eMachineState = E_MachineState.STOPPED);
stMachineStatus.bInitialising 			:= (stMachineStatus.eMachineState = E_MachineState.SYSTEM_INITIALISING);
stMachineStatus.bReadyToStart 			:= (stMachineStatus.eMachineState = E_MachineState.SYSTEM_READY_TO_START);
stMachineStatus.bAutoCycle 				:= (stMachineStatus.eMachineState = E_MachineState.SYSTEM_AUTO_CYCLE);
stMachineStatus.bStopping 				:= (stMachineStatus.eMachineState = E_MachineState.STOPPING);
stMachineStatus.bFault 					:= (stMachineStatus.eMachineState = E_MachineState.FAULT);
stMachineStatus.bManualMode 			:= (stMachineStatus.eMachineState = E_MachineState.MANUAL_MODE);
stMachineStatus.bSafety 				:= (stMachineStatus.eMachineState = E_MachineState.SAFETY);

/////////////////////////////////////////////////////////////////////////////////////FLAGS/////////////////////////////////////////////////////////////////////////////////////
stMasterCtrl.bAllStationsStopped		:= (stCamera.Status.bStopped OR NOT stMACHINE.bVisionTest ) AND (stLeakTesters.Status.bStopped OR NOT stMACHINE.bLeakTest ) AND (stHeightTests.Status.bStopped OR NOT stMACHINE.bHeightTest ) AND stProcessCylinder.Status.bStopped AND stProcessDoor.Status.bStopped AND
										   (NOT stCamera.Status.bBusy OR NOT stMACHINE.bVisionTest ) AND (NOT stLeakTesters.Status.bBusy OR NOT stMACHINE.bLeakTest ) AND (NOT stHeightTests.Status.bBusy OR NOT stMACHINE.bHeightTest ) AND NOT stProcessCylinder.Status.bBusy AND NOT stProcessDoor.Status.bBusy;
										   
stMasterCtrl.bAllStationsReady			:= (stCamera.Status.bReady OR NOT stMACHINE.bVisionTest ) AND (stLeakTesters.Status.bReady OR NOT stMACHINE.bLeakTest ) AND (stHeightTests.Status.bReady OR NOT stMACHINE.bHeightTest ) AND stProcessCylinder.Status.bReady AND stProcessDoor.Status.bReady;
END_ACTION

ACTION b_ACT_ProcessCycle:
/////////////////////////////////////////////////////////////////////////////////////UTILITIES & TRIGGERS/////////////////////////////////////////////////////////////////////////////////////
//ADD REJECT SENSOR FUNCTION. IF PART FAIL WE SHOULD WAIT UNTIL THE OPERATOR LEAVE THE FAIL PART IN THE CONTAINER
IF eCycleState = E_General_ProcessCycle.IDLE THEN
	
	bAutocycleIDLE								:= TRUE;
	
ELSE bAutocycleIDLE								:= FALSE;

END_IF

tonWaitExtendCylidner(IN := eCycleState = E_General_ProcessCycle.PROCESS_FLAGS_DEFINITIONS, PT := T#1S);
tonGettingResults( IN := eCycleState = E_General_ProcessCycle.WAIT_RESULTS, PT := T#100MS);

tonCMD_Done( IN := , PT := T#500MS);
tonSave_Data( IN :=  eCycleState = E_General_ProcessCycle.SAVE_DATA2, PT := T#500MS);
tonResetAllCMD( IN := eCycleState = E_General_ProcessCycle.RESET_ALL_CMD, PT := T#500MS);


tonExecute( IN := 	eCycleState = E_General_ProcessCycle.CLOSE_PROCESS_DOOR OR
					eCycleState = E_General_ProcessCycle.OPEN_PROCESS_DOOR OR
					eCycleState = E_General_ProcessCycle.EXTEND_PROCESS_CYLINDER OR
					eCycleState = E_General_ProcessCycle.RETRACT_PROCESS_CYLINDER OR
					eCycleState = E_General_ProcessCycle.CAMERA_INSPECTION OR
					eCycleState = E_General_ProcessCycle.LEAK_TESTS OR
					eCycleState = E_General_ProcessCycle.LEAK_TESTS_HEIGHT_TEST OR
					eCycleState = E_General_ProcessCycle.HEIGHT_TEST OR
					eCycleState = E_General_ProcessCycle.WAIT_TO_SAVE_DATA,
					PT := T#500MS);
IF (stMachineStatus.eMachineState <> E_MachineState.SYSTEM_AUTO_CYCLE) THEN
	
	eCycleState												:= E_General_ProcessCycle.RESET_ALL_CMD;

END_IF

rFirstAutoCycle( CLK := stMachineStatus.bAutoCycle);

IF (eCycleState = E_General_ProcessCycle.CAMERA_INSPECTION) OR (eCycleState = E_General_ProcessCycle.LEAK_TESTS) OR
	(eCycleState = E_General_ProcessCycle.LEAK_TESTS_HEIGHT_TEST) OR (eCycleState = E_General_ProcessCycle.HEIGHT_TEST)  THEN
			sMachineMessage						:= 'Inspection in process';

END_IF

IF stMachineStatus.eMachineState <> E_MachineState.SYSTEM_AUTO_CYCLE THEN
	
	MEMSET( destAddr := ADR(stCycleDataNest1), fillByte := 0, n := SIZEOF(stCycleDataNest1));
	MEMSET( destAddr := ADR(stCycleDataNest2), fillByte := 0, n := SIZEOF(stCycleDataNest2));

END_IF

	
/////////////////////////////////////////////////////////////////////////////////////CONDITIONS/////////////////////////////////////////////////////////////////////////////////////


bStartProcessCondition := bTwoHandsSignal AND (bPartPresentNest1 OR bPartPresentNest2);



IF rFirstAutoCycle.Q THEN
	eCycleState												:= E_General_ProcessCycle.RESET_ALL_CMD;
END_IF


CASE eCycleState OF
	
E_General_ProcessCycle.RESET_ALL_CMD:

				stProcessDoor.CMD.ProcessDoorCMD.OpenDoor						:= FALSE;
				stProcessDoor.CMD.ProcessDoorCMD.CloseDoor						:= FALSE;
				stProcessDoor.CMD.bExecute										:= FALSE;
				
				stProcessCylinder.CMD.ProcessCylinderCMD.ExtendCylinder1		:= FALSE;
				stProcessCylinder.CMD.ProcessCylinderCMD.RetractCylinder1		:= FALSE;
				stProcessCylinder.CMD.bExecute									:= FALSE;
				
				stLeakTesters.CMD.LeakTestersCMD.RunLeakTester1					:= FALSE;
				stLeakTesters.CMD.LeakTestersCMD.RunLeakTester2					:= FALSE;
				stLeakTesters.CMD.bExecute										:= FALSE;
				
				stHeightTests.CMD.HeightTest_CMD.Measurement1					:= FALSE;
				stHeightTests.CMD.HeightTest_CMD.Measurement2					:= FALSE;
				stHeightTests.CMD.bExecute										:= FALSE;
				
				stCamera.CMD.bExecute											:= FALSE;
				
				bVisionProcessDoneFlag											:= FALSE;
				
				bWriteNest1														:= FALSE;
				bWriteNest2														:= FALSE;
			
				//add reset command to reset all cycle data
				
				IF tonResetAllCMD.Q AND stMachineStatus.bAutoCycle THEN
					eCycleState								:= E_General_ProcessCycle.IDLE;						
				END_IF
	
E_General_ProcessCycle.IDLE:
		
				//start cycle
				IF bStartProcessCondition AND NOT bProcessedPart[0] AND NOT bProcessedPart[1] THEN
					
					MEMSET( destAddr := ADR(stCycleDataNest1), fillByte := 0, n := SIZEOF(stCycleDataNest1));
					MEMSET( destAddr := ADR(stCycleDataNest2), fillByte := 0, n := SIZEOF(stCycleDataNest2));
					
					bProcessedPart[0]						:= bPartPresentNest1;
					bProcessedPart[1]						:= bPartPresentNest2;
					
					eCycleState								:= E_General_ProcessCycle.CLOSE_PROCESS_DOOR;
					
				END_IF
				
				//Make sure operator remove processed part
				fProcessedPart[0]( CLK := bPartPresentNest1);
				fProcessedPart[1]( CLK := bPartPresentNest2);
				
				IF fProcessedPart[0].Q THEN
					bProcessedPart[0]						:= FALSE;
				END_IF
				
				IF fProcessedPart[1].Q THEN
					bProcessedPart[1]						:= FALSE;
				END_IF
				
				//Messages to start cycle
				IF  NOT bProcessedPart[0] AND NOT bProcessedPart[1] AND NOT bPartPresentNest1 AND NOT bPartPresentNest2  THEN
					
					sMachineMessage						:= 'Insert part to continue';
				
				ELSIF  NOT bProcessedPart[0] AND NOT bProcessedPart[1] AND ( bPartPresentNest1 OR bPartPresentNest2)  THEN
					
					sMachineMessage						:= 'trigger both safety buttons to start cycle';
				
				ELSIF bProcessedPart[0] AND NOT bProcessedPart[1] AND NOT bStartProcessCondition THEN
					
					sMachineMessage						:= 'Remove Processed part from nest 1';
					
				ELSIF NOT bProcessedPart[0] AND bProcessedPart[1] AND NOT bStartProcessCondition THEN
					
					sMachineMessage						:= 'Remove Processed part from nest 2';
					
				ELSIF bProcessedPart[0] AND bProcessedPart[1] AND NOT bStartProcessCondition THEN
					
					sMachineMessage						:= 'Remove Processed parts from both nestS';
					
				ELSE sMachineMessage						:= '';
				END_IF
				
			
E_General_ProcessCycle.CLOSE_PROCESS_DOOR:

				stProcessDoor.CMD.ProcessDoorCMD.CloseDoor	:= TRUE;
				stProcessDoor.CMD.bExecute					:= TRUE;
				
				IF tonExecute.Q THEN
					eCycleState								:= E_General_ProcessCycle.WAIT_CLOSE_PROCESS_DOOR;	
				END_IF

E_General_ProcessCycle.WAIT_CLOSE_PROCESS_DOOR:
				
				IF stProcessDoor.Status.bDone THEN
				stProcessDoor.CMD.ProcessDoorCMD.CloseDoor	:= FALSE;
				stProcessDoor.CMD.bExecute					:= FALSE;
				stProcessDoor.CMD.bAcknowledge				:= TRUE;
				eCycleState									:= E_General_ProcessCycle.PROCESS_FLAGS_DEFINITIONS;
				END_IF
				
E_General_ProcessCycle.PROCESS_FLAGS_DEFINITIONS:
					
					abLeakTesterFlag[0]						:= bPartPresentNest1;
					abLeakTesterFlag[1]						:= bPartPresentNest2;
					abHeightTestFlag[0]						:= bPartPresentNest1;
					abHeightTestFlag[1]						:= bPartPresentNest2;
				
				IF stMACHINE.bVisionTest THEN
					
					IF bVisionProcessDoneFlag THEN
						
						eCycleState							:= E_General_ProcessCycle.EXTEND_PROCESS_CYLINDER;
					ELSE eCycleState						:= E_General_ProcessCycle.CAMERA_INSPECTION;
						
					END_IF
				ELSIF tonWaitExtendCylidner.Q AND NOT stMACHINE.bVisionTest THEN

					eCycleState							:= E_General_ProcessCycle.EXTEND_PROCESS_CYLINDER;
					
				END_IF
				
				

E_General_ProcessCycle.EXTEND_PROCESS_CYLINDER:
				
						
				stProcessCylinder.CMD.ProcessCylinderCMD.ExtendCylinder1		:= TRUE;
				stProcessCylinder.CMD.bExecute		:= TRUE;
	
				IF tonExecute.Q THEN
					eCycleState								:= E_General_ProcessCycle.WAIT_EXTEND_PROCESS_CYLINDER;	
				END_IF

E_General_ProcessCycle.WAIT_EXTEND_PROCESS_CYLINDER:
			
				IF stProcessCylinder.Status.bDone THEN
					
					stProcessCylinder.CMD.ProcessCylinderCMD.ExtendCylinder1		:= FALSE;
					stProcessCylinder.CMD.bExecute			:= FALSE;
					stProcessCylinder.CMD.bAcknowledge		:= TRUE;
						
					IF stMACHINE.bHeightTest AND stMACHINE.bLeakTest THEN
						
						eCycleState							:= E_General_ProcessCycle.LEAK_TESTS_HEIGHT_TEST;	
						
					ELSIF 	stMACHINE.bHeightTest AND NOT stMACHINE.bLeakTest AND NOT stMACHINE.bVisionTest THEN
						
						eCycleState							:= E_General_ProcessCycle.HEIGHT_TEST;
					
					ELSIF 	NOT stMACHINE.bHeightTest AND stMACHINE.bLeakTest AND NOT stMACHINE.bVisionTest THEN
						
						eCycleState							:= E_General_ProcessCycle.LEAK_TESTS;
					END_IF
					
				END_IF

E_General_ProcessCycle.LEAK_TESTS_HEIGHT_TEST:
				
							
				stLeakTesters.CMD.LeakTestersCMD.RunLeakTester1						:= abLeakTesterFlag[0];
				stLeakTesters.CMD.LeakTestersCMD.RunLeakTester2						:= abLeakTesterFlag[1];
				stHeightTests.CMD.HeightTest_CMD.Measurement1						:= abHeightTestFlag[0];
				stHeightTests.CMD.HeightTest_CMD.Measurement2						:= abHeightTestFlag[1];
				stLeakTesters.CMD.bExecute					:= TRUE;
				stHeightTests.CMD.bExecute					:= TRUE;
							
				IF tonExecute.Q THEN
					eCycleState								:= E_General_ProcessCycle.WAIT_LEAK_TEST_HEIGHT_TEST;	
				END_IF

E_General_ProcessCycle.WAIT_LEAK_TEST_HEIGHT_TEST:
				
				IF (abLeakTesterFlag[0] OR abLeakTesterFlag[1]) AND (abHeightTestFlag[0] OR abHeightTestFlag[1]) THEN
					
					IF stLeakTesters.Status.bDone AND stHeightTests.Status.bDone THEN
						
						stLeakTesters.CMD.LeakTestersCMD.RunLeakTester1				:= FALSE;
						stLeakTesters.CMD.LeakTestersCMD.RunLeakTester2				:= FALSE;
						stHeightTests.CMD.HeightTest_CMD.Measurement1				:= FALSE;
						stHeightTests.CMD.HeightTest_CMD.Measurement2				:= FALSE;
						stLeakTesters.CMD.bExecute			:= FALSE;
						stHeightTests.CMD.bExecute			:= FALSE;
						stLeakTesters.CMD.bAcknowledge		:= TRUE;
						stHeightTests.CMD.bAcknowledge		:= TRUE;
						eCycleState							:= E_General_ProcessCycle.WAIT_RESULTS;
						
					END_IF
				
				ELSIF (abLeakTesterFlag[0] OR abLeakTesterFlag[1]) AND NOT (abHeightTestFlag[0] OR abHeightTestFlag[1]) THEN
					
						IF stLeakTesters.Status.bDone  THEN
						
						stLeakTesters.CMD.LeakTestersCMD.RunLeakTester1				:= FALSE;
						stLeakTesters.CMD.LeakTestersCMD.RunLeakTester2				:= FALSE;
						stLeakTesters.CMD.bExecute			:= FALSE;
						stLeakTesters.CMD.bAcknowledge		:= TRUE;
						eCycleState							:= E_General_ProcessCycle.WAIT_RESULTS;
						
					END_IF
				
				ELSIF NOT (abLeakTesterFlag[0] OR abLeakTesterFlag[1]) AND (abHeightTestFlag[0] OR abHeightTestFlag[1]) THEN
				
					IF  stHeightTests.Status.bDone THEN
						
						stHeightTests.CMD.HeightTest_CMD.Measurement1				:= FALSE;
						stHeightTests.CMD.HeightTest_CMD.Measurement2				:= FALSE;
						stHeightTests.CMD.bExecute			:= FALSE;
						stHeightTests.CMD.bAcknowledge		:= TRUE;
						eCycleState							:= E_General_ProcessCycle.WAIT_RESULTS;
					END_IF
				
				END_IF

E_General_ProcessCycle.HEIGHT_TEST:

				stHeightTests.CMD.HeightTest_CMD.Measurement1				 		:= abHeightTestFlag[0];
				stHeightTests.CMD.HeightTest_CMD.Measurement2				 		:= abHeightTestFlag[1];
				stHeightTests.CMD.bExecute					:= TRUE;
					
				IF tonExecute.Q THEN
					eCycleState								:= E_General_ProcessCycle.WAIT_HEIGHT_TEST;	
				END_IF

E_General_ProcessCycle.WAIT_HEIGHT_TEST:

				IF stHeightTests.Status.bDone THEN
					
					stHeightTests.CMD.HeightTest_CMD.Measurement1				 	:= FALSE;
					stHeightTests.CMD.HeightTest_CMD.Measurement2				 	:= FALSE;
					stHeightTests.CMD.bExecute										:= FALSE;
					stHeightTests.CMD.bAcknowledge 			:= TRUE;	
					eCycleState								:= E_General_ProcessCycle.WAIT_RESULTS;
					
				END_IF

E_General_ProcessCycle.LEAK_TESTS:

				stLeakTesters.CMD.LeakTestersCMD.RunLeakTester1						:= abHeightTestFlag[0];
				stLeakTesters.CMD.LeakTestersCMD.RunLeakTester2						:= abHeightTestFlag[1];
				stLeakTesters.CMD.bExecute					:= TRUE;
				
				IF tonExecute.Q THEN
					eCycleState								:= E_General_ProcessCycle.WAIT_LEAK_TEST;	
				END_IF

E_General_ProcessCycle.WAIT_LEAK_TEST:

				IF stLeakTesters.Status.bDone THEN
					
					stLeakTesters.CMD.bExecute										:= FALSE;
					stLeakTesters.CMD.LeakTestersCMD.RunLeakTester1				 	:= FALSE;
					stLeakTesters.CMD.LeakTestersCMD.RunLeakTester2				 	:= FALSE;
					stLeakTesters.CMD.bAcknowledge 			:= TRUE;	
					eCycleState								:= E_General_ProcessCycle.WAIT_RESULTS;
					
				END_IF
				
E_General_ProcessCycle.CAMERA_INSPECTION:
				
				stCamera.CMD.bExecute						:= TRUE;
				stCamera.CMD.CameraCMD.Inspect1				:= bPartPresentNest1;
				stCamera.CMD.CameraCMD.Inspect2				:= bPartPresentNest2;
				
				IF tonExecute.Q THEN
					eCycleState								:= E_General_ProcessCycle.WAIT_CAMERA;	
				END_IF
				
E_General_ProcessCycle.WAIT_CAMERA:

				IF stCamera.Status.bDone THEN
					
					stCamera.CMD.bExecute					:= FALSE;
					bVisionProcessDoneFlag					:= TRUE;
					stCamera.CMD.bAcknowledge				:= TRUE;
					eCycleState								:= E_General_ProcessCycle.PROCESS_FLAGS_DEFINITIONS;
				
				END_IF
				
E_General_ProcessCycle.WAIT_RESULTS:

				IF tonGettingResults.Q THEN
					
					eCycleState									:= E_General_ProcessCycle.RESULTS;
					
				END_IF


E_General_ProcessCycle.RESULTS:

				
					
					IF bProcessedPart[0] THEN
					
						IF  (stCycleDataNest1.Camera_Pass OR NOT stMACHINE.bVisionTest) AND   (stCycleDataNest1.LeakTest_Pass OR NOT stMACHINE.bLeakTest)
				 			AND   (stCycleDataNest1.HeightTest_Pass OR NOT stMACHINE.bHeightTest) THEN	
				
							stCycleDataNest1.bPass				:= TRUE;
							stCycleDataNest1.bFail				:= FALSE;
				
						ELSE stCycleDataNest1.bFail				:= TRUE;
							stCycleDataNest1.bPass				:= FALSE;
				
						END_IF
					
					END_IF
				
					IF bProcessedPart[1] THEN
					
						IF  (stCycleDataNest2.Camera_Pass OR NOT stMACHINE.bVisionTest) AND   (stCycleDataNest2.LeakTest_Pass OR NOT stMACHINE.bLeakTest)
				 			AND   (stCycleDataNest2.HeightTest_Pass OR NOT stMACHINE.bHeightTest) THEN	
				
							stCycleDataNest2.bPass				:= TRUE;
							stCycleDataNest2.bFail				:= FALSE;
				
						ELSE stCycleDataNest2.bFail				:= TRUE;
							stCycleDataNest2.bPass				:= FALSE;
				
						END_IF
					
					END_IF
					
				
				
				
				
				stCycleDataNest1.sTime						:= sSystemTime;
				stCycleDataNest1.sDate						:= sSystemDate;
				stCycleDataNest2.sTime						:= sSystemTime;
				stCycleDataNest2.sDate						:= sSystemDate;
				
				eCycleState									:= E_General_ProcessCycle.WAIT_TO_SAVE_DATA;

E_General_ProcessCycle.WAIT_TO_SAVE_DATA:
				
				IF tonExecute.Q THEN
					eCycleState								:= E_General_ProcessCycle.SAVE_DATA;	
				END_IF

E_General_ProcessCycle.SAVE_DATA:

				IF bProcessedPart[0] THEN
					
					FOR i := 199 TO 0 BY -1 DO
						aDataHistoryNest1[i+1] 						:= aDataHistoryNest1[i];
					END_FOR
				
				END_IF
				
				IF bProcessedPart[1] THEN
					
					FOR i := 199 TO 0 BY -1 DO
						aDataHistoryNest2[i+1] 						:= aDataHistoryNest2[i];
					END_FOR
				
				END_IF		
			
				eCycleState									:= E_General_ProcessCycle.SAVE_DATA2;
					
E_General_ProcessCycle.SAVE_DATA2:	
				
				
				c_ACT_SaveData();	
				
				
					
				eCycleState									:= E_General_ProcessCycle.CSV_NEST1;
				
				
E_General_ProcessCycle.CSV_NEST1:

				IF bProcessedPart[0] THEN
					
					bWriteNest1								:= TRUE;
					
					IF bCSVDone THEN
						
						eCycleState							:= E_General_ProcessCycle.CSV_NEST2;
						bWriteNest1							:= FALSE;
					END_IF
				ELSE eCycleState							:= E_General_ProcessCycle.CSV_NEST2;				
					
				END_IF
			
				
E_General_ProcessCycle.CSV_NEST2:

				IF bCSVDone THEN
					
						bWriteNest2							:= FALSE;
						eCycleState							:= E_General_ProcessCycle.RETRACT_PROCESS_CYLINDER;	
	
				END_IF

				IF bProcessedPart[1] AND  bCSVReady AND NOT bCSVDone THEN
				
						bWriteNest2							:= TRUE;

				ELSIF NOT bProcessedPart[1] THEN

						 eCycleState						:= E_General_ProcessCycle.RETRACT_PROCESS_CYLINDER;
						 
				END_IF
				
					
				
E_General_ProcessCycle.RETRACT_PROCESS_CYLINDER:
						
				stProcessCylinder.CMD.ProcessCylinderCMD.RetractCylinder1		:= TRUE;	
				stProcessCylinder.CMD.bExecute			:= TRUE;
				
				IF tonExecute.Q THEN
					eCycleState							:= E_General_ProcessCycle.WAIT_RETRACT_PROCESS_CYLINDER;	
				END_IF

E_General_ProcessCycle.WAIT_RETRACT_PROCESS_CYLINDER:

				IF 	stProcessCylinder.Status.bDone THEN
					
					stProcessCylinder.CMD.ProcessCylinderCMD.RetractCylinder1		:= FALSE;
					stProcessCylinder.CMD.bExecute		:= FALSE;
					stProcessCylinder.CMD.bAcknowledge	:= TRUE;
					
					eCycleState							:= E_General_ProcessCycle.OPEN_PROCESS_DOOR;
					
				END_IF
		
E_General_ProcessCycle.OPEN_PROCESS_DOOR:

				stProcessDoor.CMD.ProcessDoorCMD.OpenDoor							:= TRUE;
				stProcessDoor.CMD.bExecute				:= TRUE;
				
				IF tonExecute.Q THEN
					eCycleState							:= E_General_ProcessCycle.WAIT_OPEN_PROCESS_DOOR;	
				END_IF

E_General_ProcessCycle.WAIT_OPEN_PROCESS_DOOR:

				IF 	stProcessDoor.Status.bDone THEN
					
					stProcessDoor.CMD.ProcessDoorCMD.OpenDoor						:= FALSE;
					stProcessDoor.CMD.bExecute			:= FALSE;
					stProcessDoor.CMD.bAcknowledge		:= TRUE;
					
					eCycleState							:= E_General_ProcessCycle.RESET_ALL_CMD;
				END_IF
				
				
END_CASE
END_ACTION

ACTION c_ACT_SaveData:

//SAVING NEST 1 DATA
IF bProcessedPart[0] THEN
	
	stCycleDataNest1.sDistance1				:= REAL_TO_STRING(stCycleDataNest1.HeightTest_anDistancesResult[1]);
	stCycleDataNest1.sDistance2				:= REAL_TO_STRING(stCycleDataNest1.HeightTest_anDistancesResult[2]);
	stCycleDataNest1.sDistance3				:= REAL_TO_STRING(stCycleDataNest1.HeightTest_anDistancesResult[3]);
	
	stCycleDataNest1.sSetpoint1				:= REAL_TO_STRING(stCycleDataNest1.HeightTest_anSetPoint[1]);
	stCycleDataNest1.sSetpoint2				:= REAL_TO_STRING(stCycleDataNest1.HeightTest_anSetPoint[2]);
	stCycleDataNest1.sSetpoint3				:= REAL_TO_STRING(stCycleDataNest1.HeightTest_anSetPoint[3]);
	
	IF stCycleDataNest1.bPass THEN
	
		stCycleDataNest1.sGeneralResult			:= 'PASS';

	ELSIF stCycleDataNest1.bFail THEN
	
		stCycleDataNest1.sGeneralResult			:= 'FAIL';

	END_IF
	


	IF stCycleDataNest1.Camera_Pass THEN
	
		stCycleDataNest1.sCameraResult			:= 'PASS';

	ELSIF stCycleDataNest1.Camera_Fail THEN
	
		stCycleDataNest1.sCameraResult			:= 'FAIL';

	END_IF

	IF stCycleDataNest1.HeightTest_Pass THEN
	
		stCycleDataNest1.sHeightTestResult		:= 'PASS';
	
	ELSIF stCycleDataNest1.HeightTest_Fail THEN
	
		stCycleDataNest1.sHeightTestResult		:= 'FAIL';
	
	END_IF



	IF stCycleDataNest1.LeakTest_Pass THEN
	
		stCycleDataNest1.sLeakTesterResult		:= 'PASS';

	ELSIF stCycleDataNest1.LeakTest_Fail THEN
	
		stCycleDataNest1.sLeakTesterResult		:= 'FAIL';
	
	END_IF
	
	aDataHistoryNest1[0]						:= stCycleDataNest1;
	
END_IF
	

//SAVING NEST 2 DATA

IF bProcessedPart[1] THEN
	
